KUKA KRL program: MyProgram_328().src

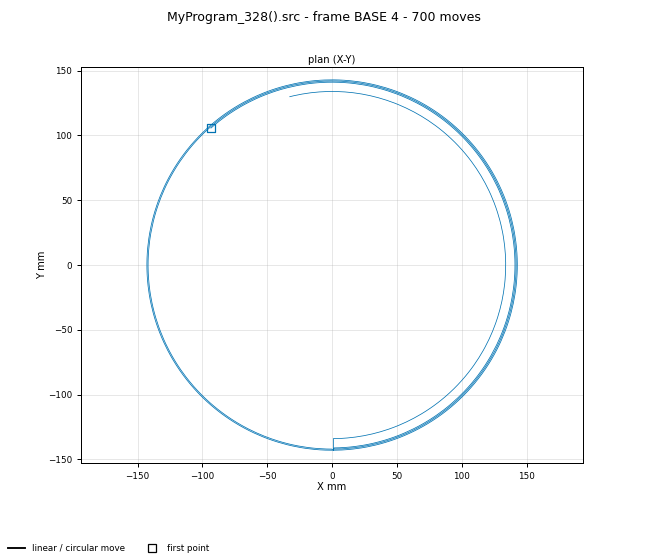
[picture p0: tool path of MyProgram_328().src in frame BASE 4, 700 of 700 moves have a stored position in this frame; points joined in program order, loops and branches not executed]
&ACCESS RVP
&REL 1
&PARAM TEMPLATE = C:\KRC\Roboter\Template\vorgabe
&PARAM EDITMASK = *
DEF MyProgram_328()
; ---- Setting reference (Base) ----
$BASE = BASE_DATA[4]

; --------------------------
; ---- Setting tool (TCP) ----
$TOOL = TOOL_DATA[3]
; --------------------------

$VEL.CP = VEL_APROX_PRINT
Startdeposition()
$VEL.CP = VEL_PRINT
LIN {X -93.4489,Y 105.68,Z 187,A 132.0784,B 2.4451,C 0.0422,E1 2.3432,E2 321.8422} C_DIS
LIN {X -90.1856,Y 108.4786,Z 187,A 130.186,B 2.4451,C 0.0397,E1 2.3473,E2 323.7515} C_DIS
LIN {X -86.5069,Y 111.4339,Z 187,A 128.2315,B 2.4451,C 0.0366,E1 2.3516,E2 325.7094} C_DIS
LIN {X -82.1262,Y 114.7007,Z 187,A 126.2266,B 2.4453,C 0.0324,E1 2.356,E2 327.6861} C_DIS
LIN {X -79.5267,Y 116.5186,Z 187,A 124.4196,B 2.4453,C 0.0324,E1 2.3603,E2 329.5564} C_DIS
LIN {X -74.9329,Y 119.5249,Z 187,A 121.6767,B 2.4453,C 0.0312,E1 2.3669,E2 332.3606} C_DIS
LIN {X -70.1382,Y 122.3996,Z 187,A 120.1865,B 2.4453,C 0.0253,E1 2.3703,E2 333.7537} C_DIS
LIN {X -67.2023,Y 124.0362,Z 187,A 118.5415,B 2.4453,C 0.0247,E1 2.3744,E2 335.4323} C_DIS
LIN {X -63.6582,Y 125.8895,Z 187,A 116.3136,B 2.4453,C 0.0253,E1 2.3802,E2 337.7328} C_DIS
LIN {X -58.7459,Y 128.2559,Z 187,A 114.739,B 2.4453,C 0.0203,E1 2.3839,E2 339.2278} C_DIS
LIN {X -55.245,Y 129.8038,Z 187,A 112.8056,B 2.4453,C 0.0204,E1 2.389,E2 341.2068} C_DIS
LIN {X -51.9085,Y 131.1741,Z 187,A 111.3758,B 2.4453,C 0.0189,E1 2.3927,E2 342.6315} C_DIS
LIN {X -45.9067,Y 133.3908,Z 187,A 108.9803,B 2.4454,C 0.016,E1 2.399,E2 345.0004} C_DIS
LIN {X -42.672,Y 134.4604,Z 187,A 107.5964,B 2.4454,C 0.015,E1 2.4027,E2 346.3836} C_DIS
LIN {X -39.1153,Y 135.5386,Z 187,A 105.5151,B 2.4454,C 0.0166,E1 2.4084,E2 348.5339} C_DIS
LIN {X -34.5458,Y 136.7738,Z 187,A 104.1224,B 2.4454,C 0.0131,E1 2.412,E2 349.8608} C_DIS
LIN {X -26.5142,Y 138.555,Z 187,A 100.5612,B 2.4454,C 0.0128,E1 2.4218,E2 353.4473} C_DIS
LIN {X -19.6263,Y 139.6976,Z 187,A 97.9243,B 2.4454,C 0.011,E1 2.4291,E2 356.0584} C_DIS
LIN {X -16.0676,Y 140.1526,Z 187,A 96.377,B 2.4454,C 0.0112,E1 2.4334,E2 357.6161} C_DIS
LIN {X -11.9745,Y 140.5601,Z 187,A 94.2351,B 2.4454,C 0.0135,E1 2.4395,E2 359.8147} C_DIS
LIN {X -7.2976,Y 140.8805,Z 187,A 92.8909,B 2.4454,C 0.0105,E1 2.4431,E2 361.0897} C_DIS
LIN {X -3.6531,Y 141.0223,Z 187,A 91.3608,B 2.4454,C 0.0109,E1 2.4474,E2 362.6252} C_DIS
LIN {X 0.7616,Y 141.0673,Z 187,A 89.5276,B 2.4454,C 0.0114,E1 2.4525,E2 364.4625} C_DIS
LIN {X 5.4307,Y 140.9647,Z 187,A 87.69,B 2.4454,C 0.0115,E1 2.4576,E2 366.2921} C_DIS
LIN {X 8.8719,Y 140.7901,Z 187,A 86.2614,B 2.4454,C 0.0122,E1 2.4616,E2 367.7237} C_DIS
LIN {X 13.2634,Y 140.4445,Z 187,A 84.4964,B 2.4454,C 0.0127,E1 2.4665,E2 369.4852} C_DIS
LIN {X 17.2396,Y 140.0128,Z 187,A 82.844,B 2.4454,C 0.0137,E1 2.4711,E2 371.1404} C_DIS
LIN {X 22.2924,Y 139.2984,Z 187,A 80.918,B 2.4454,C 0.014,E1 2.4764,E2 373.0478} C_DIS
LIN {X 24.9021,Y 138.8538,Z 187,A 79.8193,B 2.4454,C 0.0148,E1 2.4795,E2 374.1489} C_DIS
LIN {X 28.5165,Y 138.1573,Z 187,A 78.3416,B 2.4454,C 0.0158,E1 2.4835,E2 375.6241} C_DIS
LIN {X 32.2436,Y 137.3369,Z 187,A 76.8506,B 2.4454,C 0.0166,E1 2.4875,E2 377.1075} C_DIS
LIN {X 36.0345,Y 136.3894,Z 187,A 75.4608,B 2.4454,C 0.0167,E1 2.4913,E2 378.4724} C_DIS
LIN {X 38.942,Y 135.5894,Z 187,A 73.5871,B 2.4454,C 0.022,E1 2.4965,E2 380.4258} C_DIS
LIN {X 43.0848,Y 134.3286,Z 187,A 71.9887,B 2.4454,C 0.0227,E1 2.5007,E2 382.0041} C_DIS
LIN {X 46.6882,Y 133.1198,Z 187,A 70.8497,B 2.4454,C 0.0217,E1 2.5036,E2 383.093} C_DIS
LIN {X 49.6657,Y 132.037,Z 187,A 69.54,B 2.4454,C 0.0233,E1 2.507,E2 384.4053} C_DIS
LIN {X 53.4675,Y 130.5459,Z 187,A 67.9513,B 2.4454,C 0.0248,E1 2.5111,E2 385.9851} C_DIS
LIN {X 56.6566,Y 129.1935,Z 187,A 66.5966,B 2.4454,C 0.0262,E1 2.5146,E2 387.3331} C_DIS
LIN {X 59.5522,Y 127.883,Z 187,A 65.3245,B 2.4454,C 0.0278,E1 2.5178,E2 388.6026} C_DIS
LIN {X 62.4918,Y 126.472,Z 187,A 63.7782,B 2.4453,C 0.0311,E1 2.5218,E2 390.1762} C_DIS
LIN {X 65.3812,Y 125.0029,Z 187,A 62.7987,B 2.4453,C 0.0307,E1 2.5241,E2 391.1139} C_DIS
LIN {X 68.9963,Y 123.0467,Z 187,A 61.0451,B 2.4453,C 0.0337,E1 2.5284,E2 392.8779} C_DIS
LIN {X 72.7998,Y 120.8354,Z 187,A 59.2979,B 2.4452,C 0.0362,E1 2.5326,E2 394.6201} C_DIS
LIN {X 76.5853,Y 118.4724,Z 187,A 57.562,B 2.4452,C 0.0386,E1 2.5367,E2 396.3464} C_DIS
LIN {X 80.266,Y 116.0106,Z 187,A 55.7319,B 2.4452,C 0.0419,E1 2.5409,E2 398.1804} C_DIS
LIN {X 84.5184,Y 112.95,Z 187,A 53.7675,B 2.4451,C 0.0444,E1 2.5453,E2 400.1244} C_DIS
LIN {X 88.1752,Y 110.1193,Z 187,A 51.9494,B 2.4451,C 0.0474,E1 2.5493,E2 401.9351} C_DIS
LIN {X 91.0191,Y 107.7806,Z 187,A 50.5507,B 2.445,C 0.0495,E1 2.5523,E2 403.3218} C_DIS
LIN {X 94.151,Y 105.055,Z 187,A 48.609,B 2.4449,C 0.0547,E1 2.5564,E2 405.2955} C_DIS
LIN {X 97.1035,Y 102.3329,Z 187,A 47.579,B 2.4449,C 0.0535,E1 2.5584,E2 406.2504} C_DIS
LIN {X 100.7994,Y 98.6937,Z 187,A 45.3491,B 2.4448,C 0.0587,E1 2.5628,E2 408.496} C_DIS
LIN {X 103.7885,Y 95.5453,Z 187,A 43.6607,B 2.4447,C 0.0619,E1 2.566,E2 410.1752} C_DIS
LIN {X 106.7123,Y 92.2687,Z 187,A 41.9114,B 2.4446,C 0.0655,E1 2.5692,E2 411.9206} C_DIS
LIN {X 109.5484,Y 88.8835,Z 187,A 39.9522,B 2.4444,C 0.0708,E1 2.5727,E2 413.901} C_DIS
LIN {X 111.8638,Y 85.9509,Z 187,A 38.7393,B 2.4444,C 0.0719,E1 2.5747,E2 415.0758} C_DIS
LIN {X 114.5988,Y 82.2688,Z 187,A 37.005,B 2.4444,C 0.0752,E1 2.5776,E2 416.7942} C_DIS
LIN {X 117.0295,Y 78.7731,Z 187,A 35.3267,B 2.4442,C 0.0788,E1 2.5802,E2 418.4665} C_DIS
LIN {X 119.5196,Y 74.9413,Z 187,A 33.5491,B 2.4441,C 0.0827,E1 2.5829,E2 420.2346} C_DIS
LIN {X 121.8927,Y 71.0161,Z 187,A 31.7811,B 2.4439,C 0.0865,E1 2.5854,E2 421.9911} C_DIS
LIN {X 124.115,Y 67.0563,Z 187,A 30.0268,B 2.4438,C 0.0904,E1 2.5877,E2 423.7345} C_DIS
LIN {X 125.9818,Y 63.4769,Z 187,A 28.5834,B 2.4438,C 0.0929,E1 2.5895,E2 425.1532} C_DIS
LIN {X 127.4194,Y 60.5375,Z 187,A 27.2883,B 2.4436,C 0.096,E1 2.5911,E2 426.4444} C_DIS
LIN {X 128.9255,Y 57.2604,Z 187,A 25.9154,B 2.4435,C 0.099,E1 2.5927,E2 427.8061} C_DIS
LIN {X 130.3818,Y 53.8636,Z 187,A 24.5156,B 2.4433,C 0.1021,E1 2.5942,E2 429.1935} C_DIS
LIN {X 131.5987,Y 50.8162,Z 187,A 23.1723,B 2.4432,C 0.1057,E1 2.5956,E2 430.5386} C_DIS
LIN {X 132.8568,Y 47.4309,Z 187,A 21.8531,B 2.4431,C 0.1083,E1 2.5968,E2 431.8394} C_DIS
LIN {X 133.9409,Y 44.2758,Z 187,A 20.5533,B 2.4429,C 0.1115,E1 2.5979,E2 433.1327} C_DIS
LIN {X 135.1268,Y 40.5194,Z 187,A 18.45,B 2.4425,C 0.1201,E1 2.5997,E2 435.3016} C_DIS
LIN {X 136.5331,Y 35.4941,Z 187,A 17.0487,B 2.4425,C 0.1197,E1 2.6007,E2 436.6113} C_DIS
LIN {X 138.3504,Y 27.5676,Z 187,A 13.3763,B 2.4419,C 0.132,E1 2.6029,E2 440.3333} C_DIS
LIN {X 139.2135,Y 22.8091,Z 187,A 12.0869,B 2.4419,C 0.1316,E1 2.6034,E2 441.536} C_DIS
LIN {X 139.6764,Y 19.7745,Z 187,A 10.8655,B 2.4417,C 0.1349,E1 2.6039,E2 442.7547} C_DIS
LIN {X 140.0937,Y 16.5617,Z 187,A 9.6079,B 2.4416,C 0.138,E1 2.6043,E2 444.0055} C_DIS
LIN {X 140.5282,Y 12.3524,Z 187,A 7.8971,B 2.4413,C 0.1428,E1 2.6048,E2 445.7163} C_DIS
LIN {X 140.8206,Y 8.3778,Z 187,A 6.4549,B 2.4411,C 0.1458,E1 2.6051,E2 447.1363} C_DIS
LIN {X 141.0108,Y 4.0649,Z 187,A 4.8015,B 2.4409,C 0.1498,E1 2.6052,E2 448.7775} C_DIS
LIN {X 141.0688,Y 0.4654,Z 187,A 3.4438,B 2.4407,C 0.153,E1 2.6052,E2 450.1224} C_DIS
LIN {X 141.0307,Y -3.351,Z 187,A 2.023,B 2.4405,C 0.1563,E1 2.6052,E2 451.527} C_DIS
LIN {X 140.9079,Y -6.7536,Z 187,A 0.6135,B 2.4402,C 0.1604,E1 2.6051,E2 452.9409} C_DIS
LIN {X 140.6622,Y -10.7176,Z 187,A -0.8361,B 2.44,C 0.1635,E1 2.6048,E2 454.3699} C_DIS
LIN {X 140.3534,Y -14.2118,Z 187,A -2.3378,B 2.4397,C 0.1681,E1 2.6044,E2 455.8828} C_DIS
LIN {X 139.8712,Y -18.3453,Z 187,A -3.8669,B 2.4395,C 0.1715,E1 2.6039,E2 457.3917} C_DIS
LIN {X 139.3699,Y -21.831,Z 187,A -5.1458,B 2.4393,C 0.1741,E1 2.6033,E2 458.6513} C_DIS
LIN {X 138.8405,Y -24.9763,Z 187,A -6.4144,B 2.439,C 0.1775,E1 2.6027,E2 459.9172} C_DIS
LIN {X 137.7214,Y -30.5603,Z 187,A -8.657,B 2.4386,C 0.1832,E1 2.6015,E2 462.1522} C_DIS
LIN {X 136.491,Y -35.6537,Z 187,A -10.7762,B 2.4382,C 0.189,E1 2.6,E2 464.2718} C_DIS
LIN {X 135.288,Y -39.9714,Z 187,A -12.6689,B 2.4377,C 0.1946,E1 2.5985,E2 466.1754} C_DIS
LIN {X 134.115,Y -43.7528,Z 187,A -14.2718,B 2.4374,C 0.1989,E1 2.5972,E2 467.7789} C_DIS
LIN {X 132.7792,Y -47.6461,Z 187,A -15.5258,B 2.4374,C 0.1997,E1 2.596,E2 468.9781} C_DIS
LIN {X 131.393,Y -51.3455,Z 187,A -16.9763,B 2.4371,C 0.2026,E1 2.5946,E2 470.409} C_DIS
LIN {X 129.7181,Y -55.4433,Z 187,A -18.731,B 2.4367,C 0.207,E1 2.5927,E2 472.1593} C_DIS
LIN {X 126.8685,Y -61.688,Z 187,A -21.2796,B 2.4363,C 0.2121,E1 2.5898,E2 474.6779} C_DIS
LIN {X 122.4008,Y -70.1361,Z 187,A -24.8519,B 2.4356,C 0.2193,E1 2.5851,E2 478.2113} C_DIS
LIN {X 120.7802,Y -72.8911,Z 187,A -26.3212,B 2.4352,C 0.2239,E1 2.583,E2 479.705} C_DIS
LIN {X 118.2835,Y -76.8764,Z 187,A -28.2032,B 2.4348,C 0.2283,E1 2.5801,E2 481.5846} C_DIS
LIN {X 115.9942,Y -80.2896,Z 187,A -29.7454,B 2.4345,C 0.2312,E1 2.5777,E2 483.1109} C_DIS
LIN {X 112.5091,Y -85.1039,Z 187,A -31.8029,B 2.4343,C 0.2339,E1 2.5744,E2 485.1217} C_DIS
LIN {X 110.5589,Y -87.6229,Z 187,A -33.2922,B 2.4338,C 0.2385,E1 2.5718,E2 486.6387} C_DIS
LIN {X 107.5329,Y -91.3106,Z 187,A -35.3251,B 2.4333,C 0.2436,E1 2.5681,E2 488.6862} C_DIS
LIN {X 105.2436,Y -93.9402,Z 187,A -36.5934,B 2.4331,C 0.2455,E1 2.5658,E2 489.9354} C_DIS
LIN {X 101.7183,Y -97.7471,Z 187,A -39.1489,B 2.4323,C 0.2536,E1 2.5608,E2 492.5536} C_DIS
LIN {X 97.3968,Y -102.0531,Z 187,A -40.896,B 2.4323,C 0.2528,E1 2.5574,E2 494.203} C_DIS
LIN {X 92.0106,Y -106.9346,Z 187,A -43.3577,B 2.4322,C 0.2547,E1 2.5525,E2 496.5995} C_DIS
LIN {X 88.677,Y -109.7149,Z 187,A -45.5587,B 2.4314,C 0.2615,E1 2.5476,E2 498.8623} C_DIS
LIN {X 86.1521,Y -111.7089,Z 187,A -47.2607,B 2.4309,C 0.267,E1 2.5437,E2 500.6194} C_DIS
LIN {X 81.5208,Y -115.132,Z 187,A -48.6174,B 2.4312,C 0.2635,E1 2.5409,E2 501.8429} C_DIS
LIN {X 79.0495,Y -116.8424,Z 187,A -50.4786,B 2.4305,C 0.2706,E1 2.5364,E2 503.7933} C_DIS
LIN {X 75.3103,Y -119.2862,Z 187,A -51.9221,B 2.4305,C 0.2707,E1 2.5331,E2 505.1872} C_DIS
LIN {X 71.0161,Y -121.8927,Z 187,A -53.8333,B 2.4302,C 0.2729,E1 2.5285,E2 507.0822} C_DIS
LIN {X 67.0764,Y -124.1042,Z 187,A -55.6212,B 2.4299,C 0.2753,E1 2.5242,E2 508.8648} C_DIS
LIN {X 63.1985,Y -126.1233,Z 187,A -57.2403,B 2.4298,C 0.2767,E1 2.5202,E2 510.4636} C_DIS
LIN {X 56.1606,Y -129.408,Z 187,A -60.0745,B 2.4296,C 0.2786,E1 2.5131,E2 513.2555} C_DIS
LIN {X 51.9792,Y -131.1459,Z 187,A -62.1004,B 2.4291,C 0.2822,E1 2.5078,E2 515.3088} C_DIS
LIN {X 48.5186,Y -132.4646,Z 187,A -63.7676,B 2.4288,C 0.2851,E1 2.5034,E2 516.9996} C_DIS
LIN {X 44.3169,Y -133.9273,Z 187,A -65.3456,B 2.4288,C 0.2854,E1 2.4993,E2 518.5469} C_DIS
LIN {X 40.4578,Y -135.1456,Z 187,A -67.0119,B 2.4285,C 0.2873,E1 2.4948,E2 520.2175} C_DIS
LIN {X 36.0324,Y -136.39,Z 187,A -68.8114,B 2.4284,C 0.2885,E1 2.49,E2 522.0087} C_DIS
LIN {X 31.8028,Y -137.438,Z 187,A -70.552,B 2.4282,C 0.2898,E1 2.4852,E2 523.7464} C_DIS
LIN {X 27.8459,Y -138.2937,Z 187,A -72.1648,B 2.4282,C 0.2909,E1 2.4808,E2 525.3558} C_DIS
LIN {X 24.2043,Y -138.9786,Z 187,A -74.473,B 2.4274,C 0.2972,E1 2.4742,E2 527.7761} C_DIS
LIN {X 17.7076,Y -139.9548,Z 187,A -76.3709,B 2.4278,C 0.2937,E1 2.4692,E2 529.5691} C_DIS
LIN {X 13.6314,Y -140.4091,Z 187,A -77.9481,B 2.4278,C 0.2939,E1 2.4648,E2 531.1348} C_DIS
LIN {X 9.8054,Y -140.7288,Z 187,A -79.5631,B 2.4276,C 0.2949,E1 2.4603,E2 532.7584} C_DIS
LIN {X 5.6236,Y -140.9572,Z 187,A -81.1799,B 2.4276,C 0.2949,E1 2.4558,E2 534.3642} C_DIS
LIN {X 1.6647,Y -141.0612,Z 187,A -82.8613,B 2.4276,C 0.2958,E1 2.4511,E2 536.0567} C_DIS
LIN {X 1.6647,Y -141.0612,Z 187,A -82.8613,B 2.4276,C 0.2958,E1 2.4511,E2 536.0567} C_DIS
Enddeposition()
LIN {X 0.9996,Y -141.963,Z 187,A -82.7924,B 2.4278,C 0.2951,E1 2.4515,E2 535.9704} C_DIS
Startdeposition()
$VEL.CP = VEL_PRINT
LIN {X 3.7682,Y -141.9191,Z 187,A -81.2714,B 2.4281,C 0.2923,E1 2.4559,E2 534.3919} C_DIS
LIN {X 7.2589,Y -141.7833,Z 187,A -79.8823,B 2.4281,C 0.292,E1 2.4598,E2 533.005} C_DIS
LIN {X 11.0857,Y -141.5374,Z 187,A -78.324,B 2.4282,C 0.2913,E1 2.4641,E2 531.4445} C_DIS
LIN {X 14.9868,Y -141.1758,Z 187,A -76.8976,B 2.4282,C 0.2915,E1 2.468,E2 530.039} C_DIS
LIN {X 17.882,Y -140.8393,Z 187,A -75.3634,B 2.4285,C 0.2885,E1 2.4724,E2 528.4534} C_DIS
LIN {X 23.036,Y -140.0878,Z 187,A -73.5358,B 2.4285,C 0.2891,E1 2.4774,E2 526.6635} C_DIS
LIN {X 26.407,Y -139.4914,Z 187,A -72.2818,B 2.4285,C 0.289,E1 2.4808,E2 525.4268} C_DIS
LIN {X 29.7911,Y -138.8079,Z 187,A -70.7974,B 2.4287,C 0.2873,E1 2.4849,E2 523.9287} C_DIS
LIN {X 32.6858,Y -138.1561,Z 187,A -69.705,B 2.4287,C 0.287,E1 2.4878,E2 522.8505} C_DIS
LIN {X 36.0579,Y -137.3143,Z 187,A -68.3438,B 2.4288,C 0.2861,E1 2.4915,E2 521.4943} C_DIS
LIN {X 39.1204,Y -136.4746,Z 187,A -66.8529,B 2.4291,C 0.2834,E1 2.4956,E2 519.973} C_DIS
LIN {X 43.2015,Y -135.2357,Z 187,A -65.3089,B 2.4291,C 0.2829,E1 2.4997,E2 518.4528} C_DIS
LIN {X 47.5675,Y -133.7639,Z 187,A -63.4225,B 2.4295,C 0.2807,E1 2.5047,E2 516.5614} C_DIS
LIN {X 51.1458,Y -132.4359,Z 187,A -62.0665,B 2.4295,C 0.2803,E1 2.5082,E2 515.2304} C_DIS
LIN {X 53.7562,Y -131.3996,Z 187,A -60.7366,B 2.4298,C 0.2774,E1 2.5117,E2 513.8721} C_DIS
LIN {X 56.7664,Y -130.1262,Z 187,A -59.2192,B 2.4302,C 0.2743,E1 2.5156,E2 512.3256} C_DIS
LIN {X 60.3683,Y -128.4969,Z 187,A -57.8944,B 2.4302,C 0.2741,E1 2.5189,E2 511.0381} C_DIS
LIN {X 63.9328,Y -126.7593,Z 187,A -56.289,B 2.4305,C 0.2718,E1 2.5229,E2 509.4308} C_DIS
LIN {X 68.2838,Y -124.4711,Z 187,A -54.4459,B 2.4307,C 0.27,E1 2.5274,E2 507.6063} C_DIS
LIN {X 71.2977,Y -122.7693,Z 187,A -52.7218,B 2.4312,C 0.2653,E1 2.5317,E2 505.8348} C_DIS
LIN {X 75.1294,Y -120.4624,Z 187,A -50.6328,B 2.4317,C 0.2601,E1 2.5367,E2 503.7041} C_DIS
LIN {X 80.5629,Y -116.8987,Z 187,A -49.0053,B 2.4314,C 0.2635,E1 2.5402,E2 502.2154} C_DIS
LIN {X 84.7135,Y -113.9265,Z 187,A -46.767,B 2.4319,C 0.2584,E1 2.5453,E2 499.9506} C_DIS
LIN {X 88.639,Y -110.9,Z 187,A -44.9104,B 2.4322,C 0.2559,E1 2.5494,E2 498.1126} C_DIS
LIN {X 92.22,Y -107.9408,Z 187,A -43.2469,B 2.4324,C 0.254,E1 2.5529,E2 496.4773} C_DIS
LIN {X 95.9781,Y -104.6128,Z 187,A -40.9372,B 2.433,C 0.2476,E1 2.5577,E2 494.1263} C_DIS
LIN {X 98.5673,Y -102.1771,Z 187,A -39.7798,B 2.4331,C 0.247,E1 2.56,E2 493.0066} C_DIS
LIN {X 101.6156,Y -99.1464,Z 187,A -38.1008,B 2.4334,C 0.2438,E1 2.5633,E2 491.3341} C_DIS
LIN {X 104.7827,Y -95.7932,Z 187,A -36.4189,B 2.4337,C 0.2413,E1 2.5664,E2 489.6758} C_DIS
LIN {X 107.0817,Y -93.2155,Z 187,A -34.6604,B 2.4343,C 0.2352,E1 2.5698,E2 487.8652} C_DIS
LIN {X 109.8305,Y -89.9605,Z 187,A -33.3443,B 2.4343,C 0.2347,E1 2.572,E2 486.6041} C_DIS
LIN {X 112.7503,Y -86.2727,Z 187,A -31.4726,B 2.4347,C 0.2306,E1 2.5752,E2 484.7347} C_DIS
LIN {X 115.5827,Y -82.4395,Z 187,A -29.7495,B 2.435,C 0.2278,E1 2.578,E2 483.0379} C_DIS
LIN {X 118.0467,Y -78.8707,Z 187,A -28.0529,B 2.4353,C 0.2241,E1 2.5807,E2 481.3474} C_DIS
LIN {X 120.4789,Y -75.103,Z 187,A -26.318,B 2.4357,C 0.2203,E1 2.5832,E2 479.6215} C_DIS
LIN {X 122.8161,Y -71.2168,Z 187,A -24.7349,B 2.4359,C 0.2179,E1 2.5854,E2 478.0712} C_DIS
LIN {X 125.4596,Y -66.4467,Z 187,A -22.5256,B 2.4364,C 0.2123,E1 2.5884,E2 475.859} C_DIS
LIN {X 127.0868,Y -63.2792,Z 187,A -21.155,B 2.4366,C 0.2092,E1 2.5901,E2 474.4964} C_DIS
LIN {X 128.6491,Y -60.039,Z 187,A -19.6284,B 2.437,C 0.2048,E1 2.592,E2 472.9584} C_DIS
LIN {X 130.7091,Y -55.4144,Z 187,A -17.9178,B 2.4372,C 0.2024,E1 2.5938,E2 471.2921} C_DIS
LIN {X 132.1546,Y -51.8693,Z 187,A -16.3795,B 2.4376,C 0.1984,E1 2.5954,E2 469.7535} C_DIS
LIN {X 134.6378,Y -45.0306,Z 187,A -13.8601,B 2.4379,C 0.1943,E1 2.5977,E2 467.2891} C_DIS
LIN {X 135.6936,Y -41.7415,Z 187,A -12.2862,B 2.4383,C 0.1889,E1 2.5991,E2 465.6896} C_DIS
LIN {X 136.6561,Y -38.4741,Z 187,A -10.6448,B 2.4388,C 0.1828,E1 2.6004,E2 464.0107} C_DIS
LIN {X 137.6676,Y -34.6814,Z 187,A -9.4864,B 2.4388,C 0.1822,E1 2.6011,E2 462.9095} C_DIS
LIN {X 138.626,Y -30.6336,Z 187,A -7.7706,B 2.4392,C 0.1773,E1 2.6022,E2 461.1875} C_DIS
LIN {X 139.3977,Y -26.8975,Z 187,A -6.4337,B 2.4394,C 0.1748,E1 2.6029,E2 459.877} C_DIS
LIN {X 140.0385,Y -23.3314,Z 187,A -5.0733,B 2.4396,C 0.1717,E1 2.6035,E2 458.5294} C_DIS
LIN {X 140.6556,Y -19.2805,Z 187,A -3.4323,B 2.4399,C 0.1672,E1 2.6042,E2 456.8891} C_DIS
LIN {X 141.1483,Y -15.2421,Z 187,A -1.975,B 2.4401,C 0.1642,E1 2.6046,E2 455.4556} C_DIS
LIN {X 141.4775,Y -11.8026,Z 187,A -0.6039,B 2.4403,C 0.1605,E1 2.605,E2 454.0868} C_DIS
LIN {X 141.7785,Y -7.3542,Z 187,A 1.0076,B 2.4406,C 0.1571,E1 2.6053,E2 452.4994} C_DIS
LIN {X 141.9161,Y -3.8773,Z 187,A 2.4541,B 2.4408,C 0.1528,E1 2.6053,E2 451.0464} C_DIS
LIN {X 141.9682,Y 0.508,Z 187,A 4.1072,B 2.4411,C 0.1489,E1 2.6054,E2 449.4078} C_DIS
LIN {X 141.9065,Y 4.2199,Z 187,A 5.523,B 2.4413,C 0.1454,E1 2.6054,E2 448.0023} C_DIS
LIN {X 141.7092,Y 8.5854,Z 187,A 7.0861,B 2.4415,C 0.1422,E1 2.6051,E2 446.465} C_DIS
LIN {X 141.4746,Y 11.8375,Z 187,A 8.4459,B 2.4417,C 0.1381,E1 2.6048,E2 445.0986} C_DIS
LIN {X 141.0538,Y 16.1086,Z 187,A 10.1489,B 2.442,C 0.1336,E1 2.6043,E2 443.3986} C_DIS
LIN {X 140.5408,Y 20.0852,Z 187,A 11.5878,B 2.4421,C 0.1306,E1 2.6038,E2 441.9826} C_DIS
LIN {X 139.991,Y 23.6157,Z 187,A 13.0025,B 2.4423,C 0.1269,E1 2.6031,E2 440.5708} C_DIS
LIN {X 139.0168,Y 28.8045,Z 187,A 15.0092,B 2.4426,C 0.1221,E1 2.602,E2 438.5795} C_DIS
LIN {X 138.0808,Y 32.9981,Z 187,A 16.6182,B 2.4427,C 0.1184,E1 2.601,E2 436.9862} C_DIS
LIN {X 137.2031,Y 36.4748,Z 187,A 17.9412,B 2.4429,C 0.1155,E1 2.6001,E2 435.679} C_DIS
LIN {X 136.3607,Y 39.5094,Z 187,A 19.3511,B 2.4431,C 0.1109,E1 2.599,E2 434.25} C_DIS
LIN {X 134.8365,Y 44.4339,Z 187,A 21.0397,B 2.4431,C 0.1087,E1 2.5976,E2 432.6123} C_DIS
LIN {X 133.687,Y 47.7808,Z 187,A 22.431,B 2.4433,C 0.1052,E1 2.5964,E2 431.2252} C_DIS
LIN {X 132.5412,Y 50.8749,Z 187,A 23.6494,B 2.4435,C 0.1026,E1 2.5952,E2 430.0213} C_DIS
LIN {X 131.0962,Y 54.4875,Z 187,A 25.1666,B 2.4436,C 0.0989,E1 2.5936,E2 428.5103} C_DIS
LIN {X 129.7867,Y 57.5383,Z 187,A 26.5247,B 2.4438,C 0.0953,E1 2.5921,E2 427.1493} C_DIS
LIN {X 128.2461,Y 60.8941,Z 187,A 27.9417,B 2.4438,C 0.0921,E1 2.5904,E2 425.7414} C_DIS
LIN {X 126.7611,Y 63.9292,Z 187,A 29.2664,B 2.444,C 0.0889,E1 2.5888,E2 424.4213} C_DIS
LIN {X 124.8445,Y 67.5992,Z 187,A 30.9033,B 2.4441,C 0.085,E1 2.5866,E2 422.7884} C_DIS
LIN {X 122.644,Y 71.514,Z 187,A 32.6528,B 2.4443,C 0.0811,E1 2.5842,E2 421.0466} C_DIS
LIN {X 120.3764,Y 75.2676,Z 187,A 34.287,B 2.4443,C 0.0779,E1 2.5818,E2 419.4295} C_DIS
LIN {X 117.9973,Y 78.9446,Z 187,A 35.9633,B 2.4445,C 0.0744,E1 2.5793,E2 417.7645} C_DIS
LIN {X 115.4017,Y 82.6927,Z 187,A 37.7059,B 2.4445,C 0.0709,E1 2.5765,E2 416.0342} C_DIS
LIN {X 112.7821,Y 86.2311,Z 187,A 39.4389,B 2.4447,C 0.0672,E1 2.5736,E2 414.3063} C_DIS
LIN {X 110.0375,Y 89.7071,Z 187,A 41.1027,B 2.4447,C 0.0641,E1 2.5707,E2 412.6582} C_DIS
LIN {X 107.4472,Y 92.794,Z 187,A 42.6833,B 2.4449,C 0.0609,E1 2.5678,E2 411.0833} C_DIS
LIN {X 104.407,Y 96.2019,Z 187,A 44.4152,B 2.4449,C 0.0578,E1 2.5646,E2 409.3654} C_DIS
LIN {X 101.4157,Y 99.3502,Z 187,A 46.1356,B 2.445,C 0.0544,E1 2.5613,E2 407.6489} C_DIS
LIN {X 98.1632,Y 102.5651,Z 187,A 47.6842,B 2.445,C 0.0529,E1 2.5583,E2 406.1382} C_DIS
LIN {X 95.5959,Y 104.9624,Z 187,A 49.2623,B 2.4451,C 0.0489,E1 2.555,E2 404.5394} C_DIS
LIN {X 92.3606,Y 107.8205,Z 187,A 50.9361,B 2.4451,C 0.046,E1 2.5515,E2 402.8743} C_DIS
LIN {X 89.3733,Y 110.3091,Z 187,A 52.4532,B 2.4452,C 0.0435,E1 2.5482,E2 401.3637} C_DIS
LIN {X 85.9012,Y 113.0344,Z 187,A 54.1813,B 2.4452,C 0.0406,E1 2.5444,E2 399.6424} C_DIS
LIN {X 82.3582,Y 115.6409,Z 187,A 55.8678,B 2.4453,C 0.0382,E1 2.5406,E2 397.9673} C_DIS
LIN {X 78.849,Y 118.0612,Z 187,A 57.5179,B 2.4453,C 0.0358,E1 2.5368,E2 396.3261} C_DIS
LIN {X 75.3466,Y 120.3273,Z 187,A 59.1625,B 2.4453,C 0.0334,E1 2.5329,E2 394.6866} C_DIS
LIN {X 71.5652,Y 122.614,Z 187,A 60.9314,B 2.4454,C 0.0307,E1 2.5287,E2 392.9196} C_DIS
LIN {X 67.5831,Y 124.8533,Z 187,A 62.5878,B 2.4454,C 0.0293,E1 2.5247,E2 391.2871} C_DIS
LIN {X 65.0121,Y 126.2098,Z 187,A 63.8486,B 2.4454,C 0.027,E1 2.5215,E2 390.0153} C_DIS
LIN {X 61.8211,Y 127.8032,Z 187,A 65.2354,B 2.4454,C 0.0254,E1 2.5181,E2 388.6354} C_DIS
LIN {X 58.2382,Y 129.4737,Z 187,A 66.5719,B 2.4454,C 0.0251,E1 2.5147,E2 387.3317} C_DIS
LIN {X 55.7537,Y 130.5641,Z 187,A 67.8714,B 2.4455,C 0.0224,E1 2.5113,E2 386.0066} C_DIS
LIN {X 51.9672,Y 132.1165,Z 187,A 69.3282,B 2.4455,C 0.0217,E1 2.5076,E2 384.5747} C_DIS
LIN {X 48.52,Y 133.4205,Z 187,A 70.6667,B 2.4455,C 0.021,E1 2.5042,E2 383.2552} C_DIS
LIN {X 42.9455,Y 135.3175,Z 187,A 73.8187,B 2.4455,C 0.0135,E1 2.4955,E2 380.0055} C_DIS
LIN {X 37.6109,Y 136.8975,Z 187,A 75.6157,B 2.4455,C 0.0144,E1 2.4908,E2 378.2661} C_DIS
LIN {X 32.6143,Y 138.1733,Z 187,A 77.409,B 2.4455,C 0.0144,E1 2.4861,E2 376.5098} C_DIS
LIN {X 29.0269,Y 138.9716,Z 187,A 78.9989,B 2.4455,C 0.0127,E1 2.4817,E2 374.9068} C_DIS
LIN {X 25.5257,Y 139.6561,Z 187,A 80.1674,B 2.4455,C 0.0134,E1 2.4786,E2 373.7728} C_DIS
LIN {X 22.4562,Y 140.1835,Z 187,A 81.7525,B 2.4455,C 0.0106,E1 2.4741,E2 372.1469} C_DIS
LIN {X 17.6812,Y 140.8656,Z 187,A 83.5823,B 2.4455,C 0.0103,E1 2.469,E2 370.3325} C_DIS
LIN {X 13.7164,Y 141.3048,Z 187,A 85.0418,B 2.4455,C 0.0105,E1 2.465,E2 368.8924} C_DIS
LIN {X 10.2703,Y 141.597,Z 187,A 86.3842,B 2.4455,C 0.0102,E1 2.4613,E2 367.5571} C_DIS
LIN {X 7.1493,Y 141.7888,Z 187,A 87.7138,B 2.4455,C 0.0094,E1 2.4576,E2 366.2196} C_DIS
LIN {X 2.9737,Y 141.9392,Z 187,A 89.4396,B 2.4455,C 0.0088,E1 2.4527,E2 364.4895} C_DIS
LIN {X -0.7732,Y 141.9669,Z 187,A 90.954,B 2.4455,C 0.0085,E1 2.4485,E2 362.9754} C_DIS
LIN {X -5.5262,Y 141.8614,Z 187,A 92.7703,B 2.4455,C 0.009,E1 2.4434,E2 361.1728} C_DIS
LIN {X -9.8597,Y 141.6269,Z 187,A 94.4629,B 2.4455,C 0.0093,E1 2.4387,E2 359.4883} C_DIS
LIN {X -13.6559,Y 141.3106,Z 187,A 96.1386,B 2.4455,C 0.0087,E1 2.434,E2 357.796} C_DIS
LIN {X -18.1954,Y 140.7982,Z 187,A 97.9544,B 2.4455,C 0.0091,E1 2.429,E2 355.9846} C_DIS
LIN {X -22.019,Y 140.2512,Z 187,A 99.9681,B 2.4455,C 0.0072,E1 2.4233,E2 353.9145} C_DIS
LIN {X -26.3023,Y 139.5114,Z 187,A 101.2219,B 2.4455,C 0.0104,E1 2.42,E2 352.7246} C_DIS
LIN {X -29.1917,Y 138.9373,Z 187,A 102.516,B 2.4455,C 0.0104,E1 2.4164,E2 351.418} C_DIS
LIN {X -32.657,Y 138.163,Z 187,A 104.0144,B 2.4455,C 0.0107,E1 2.4123,E2 349.9122} C_DIS
LIN {X -36.3809,Y 137.2281,Z 187,A 105.8057,B 2.4455,C 0.0104,E1 2.4074,E2 348.0913} C_DIS
LIN {X -39.7779,Y 136.2821,Z 187,A 106.9762,B 2.4455,C 0.0125,E1 2.4043,E2 346.9533} C_DIS
LIN {X -43.7202,Y 135.07,Z 187,A 108.7525,B 2.4455,C 0.0131,E1 2.3995,E2 345.164} C_DIS
LIN {X -50.6272,Y 132.6373,Z 187,A 111.7286,B 2.4455,C 0.0154,E1 2.3917,E2 342.1872} C_DIS
LIN {X -54.3321,Y 131.1611,Z 187,A 113.1961,B 2.4455,C 0.0175,E1 2.388,E2 340.7384} C_DIS
LIN {X -57.7103,Y 129.7098,Z 187,A 114.7724,B 2.4455,C 0.0186,E1 2.3839,E2 339.1514} C_DIS
LIN {X -60.7714,Y 128.3047,Z 187,A 116.4131,B 2.4455,C 0.0188,E1 2.3797,E2 337.4761} C_DIS
LIN {X -63.6843,Y 126.8858,Z 187,A 117.5622,B 2.4455,C 0.021,E1 2.3768,E2 336.348} C_DIS
LIN {X -67.4063,Y 124.9482,Z 187,A 119.3288,B 2.4455,C 0.0227,E1 2.3724,E2 334.5732} C_DIS
LIN {X -70.536,Y 123.2085,Z 187,A 120.9137,B 2.4455,C 0.0239,E1 2.3685,E2 332.9716} C_DIS
LIN {X -74.8507,Y 120.6359,Z 187,A 122.9065,B 2.4455,C 0.0268,E1 2.3638,E2 330.9845} C_DIS
LIN {X -78.7501,Y 118.1272,Z 187,A 124.8088,B 2.4455,C 0.0293,E1 2.3593,E2 329.0797} C_DIS
LIN {X -82.3891,Y 115.6187,Z 187,A 126.694,B 2.4455,C 0.0316,E1 2.355,E2 327.1828} C_DIS
LIN {X -86.1482,Y 112.8455,Z 187,A 128.5791,B 2.4454,C 0.0346,E1 2.3508,E2 325.299} C_DIS
LIN {X -89.5032,Y 110.2042,Z 187,A 130.4211,B 2.4454,C 0.0371,E1 2.3467,E2 323.4433} C_DIS
LIN {X -93.0071,Y 107.2636,Z 187,A 132.1594,B 2.4453,C 0.0406,E1 2.3431,E2 321.7199} C_DIS
LIN {X -95.6368,Y 104.9252,Z 187,A 133.7545,B 2.4453,C 0.0426,E1 2.3397,E2 320.1036} C_DIS
LIN {X -98.7853,Y 101.966,Z 187,A 135.5669,B 2.4452,C 0.0456,E1 2.336,E2 318.2837} C_DIS
LIN {X -101.5357,Y 99.2279,Z 187,A 137.2404,B 2.4452,C 0.0482,E1 2.3327,E2 316.5978} C_DIS
LIN {X -104.3309,Y 96.2847,Z 187,A 139.0136,B 2.4451,C 0.051,E1 2.3293,E2 314.8086} C_DIS
LIN {X -107.6788,Y 92.5251,Z 187,A 141.0456,B 2.445,C 0.0552,E1 2.3256,E2 312.778} C_DIS
LIN {X -110.2091,Y 89.4973,Z 187,A 142.77,B 2.445,C 0.0581,E1 2.3225,E2 311.0379} C_DIS
LIN {X -113.0558,Y 85.8731,Z 187,A 144.4305,B 2.4448,C 0.0627,E1 2.3197,E2 309.4042} C_DIS
LIN {X -115.947,Y 81.9263,Z 187,A 146.6612,B 2.4448,C 0.0664,E1 2.316,E2 307.1423} C_DIS
LIN {X -117.5624,Y 79.5907,Z 187,A 147.9369,B 2.4446,C 0.0686,E1 2.3139,E2 305.8508} C_DIS
LIN {X -119.9532,Y 75.94,Z 187,A 149.8296,B 2.4446,C 0.0723,E1 2.311,E2 303.9425} C_DIS
LIN {X -122.4267,Y 71.8841,Z 187,A 151.805,B 2.4444,C 0.0767,E1 2.3082,E2 301.961} C_DIS
LIN {X -124.6117,Y 68.026,Z 187,A 153.5249,B 2.4443,C 0.0812,E1 2.3059,E2 300.2514} C_DIS
LIN {X -126.197,Y 65.0371,Z 187,A 155.1662,B 2.4442,C 0.0838,E1 2.3037,E2 298.5755} C_DIS
LIN {X -127.8502,Y 61.7227,Z 187,A 156.6552,B 2.444,C 0.0875,E1 2.3019,E2 297.0882} C_DIS
LIN {X -129.4019,Y 58.3988,Z 187,A 158.1848,B 2.444,C 0.0912,E1 2.3001,E2 295.5534} C_DIS
LIN {X -130.9979,Y 54.723,Z 187,A 159.7031,B 2.4437,C 0.0956,E1 2.2984,E2 294.0491} C_DIS
LIN {X -132.2138,Y 51.7171,Z 187,A 161.3539,B 2.4437,C 0.0981,E1 2.2967,E2 292.3548} C_DIS
LIN {X -133.6411,Y 47.9081,Z 187,A 162.9786,B 2.4435,C 0.1024,E1 2.2951,E2 290.7336} C_DIS
LIN {X -134.6713,Y 44.9302,Z 187,A 164.4028,B 2.4433,C 0.1054,E1 2.2938,E2 289.2904} C_DIS
LIN {X -135.768,Y 41.4984,Z 187,A 165.9228,B 2.4432,C 0.1091,E1 2.2926,E2 287.7628} C_DIS
LIN {X -136.7761,Y 38.0449,Z 187,A 167.4839,B 2.443,C 0.1127,E1 2.2914,E2 286.1885} C_DIS
LIN {X -137.9061,Y 33.7228,Z 187,A 169.4221,B 2.4428,C 0.1173,E1 2.29,E2 284.2339} C_DIS
LIN {X -139.805,Y 24.6939,Z 187,A 172.8607,B 2.4422,C 0.1283,E1 2.2881,E2 280.8355} C_DIS
LIN {X -140.4475,Y 20.7386,Z 187,A 175.1058,B 2.4421,C 0.1312,E1 2.2871,E2 278.5092} C_DIS
LIN {X -140.8929,Y 17.4571,Z 187,A 176.5678,B 2.4419,C 0.1346,E1 2.2865,E2 277.0315} C_DIS
LIN {X -141.3104,Y 13.6576,Z 187,A 177.9513,B 2.4416,C 0.1393,E1 2.2862,E2 275.6699} C_DIS
LIN {X -141.5316,Y 11.1627,Z 187,A 179.2339,B 2.4416,C 0.1414,E1 2.2859,E2 274.3522} C_DIS
LIN {X -141.7436,Y 8.0273,Z 187,A -179.3993,B 2.4413,C 0.1448,E1 2.2856,E2 272.9731} C_DIS
LIN {X -141.9294,Y 3.3985,Z 187,A -177.394,B 2.441,C 0.1497,E1 2.2854,E2 270.9508} C_DIS
LIN {X -141.9653,Y -1.0663,Z 187,A -175.5455,B 2.4407,C 0.1546,E1 2.2854,E2 269.0972} C_DIS
LIN {X -141.8675,Y -5.3683,Z 187,A -173.8566,B 2.4404,C 0.1596,E1 2.2856,E2 267.4158} C_DIS
LIN {X -141.6419,Y -9.655,Z 187,A -171.8203,B 2.4401,C 0.1637,E1 2.2859,E2 265.34} C_DIS
LIN {X -141.1197,Y -15.5075,Z 187,A -169.3476,B 2.4397,C 0.17,E1 2.2866,E2 262.8551} C_DIS
LIN {X -140.5823,Y -19.795,Z 187,A -167.6331,B 2.4393,C 0.175,E1 2.2872,E2 261.1456} C_DIS
LIN {X -140.0836,Y -23.0608,Z 187,A -166.1046,B 2.4391,C 0.1781,E1 2.2879,E2 259.5915} C_DIS
LIN {X -138.9037,Y -29.3472,Z 187,A -163.3411,B 2.4386,C 0.1848,E1 2.2894,E2 256.8049} C_DIS
LIN {X -138.0745,Y -33.0242,Z 187,A -161.768,B 2.4383,C 0.1887,E1 2.2904,E2 255.2255} C_DIS
LIN {X -137.1868,Y -36.536,Z 187,A -160.1642,B 2.438,C 0.1923,E1 2.2915,E2 253.6032} C_DIS
LIN {X -136.0472,Y -40.5803,Z 187,A -158.3514,B 2.4377,C 0.1965,E1 2.2929,E2 251.7754} C_DIS
LIN {X -134.8365,Y -44.4339,Z 187,A -156.6444,B 2.4374,C 0.2006,E1 2.2944,E2 250.0587} C_DIS
LIN {X -133.862,Y -47.2942,Z 187,A -155.2575,B 2.4371,C 0.2034,E1 2.2957,E2 248.6496} C_DIS
LIN {X -132.4832,Y -51.0242,Z 187,A -153.8732,B 2.4367,C 0.2081,E1 2.297,E2 247.296} C_DIS
LIN {X -131.1245,Y -54.4197,Z 187,A -152.1482,B 2.4365,C 0.2112,E1 2.2989,E2 245.5377} C_DIS
LIN {X -129.7648,Y -57.5874,Z 187,A -150.8505,B 2.4361,C 0.215,E1 2.3003,E2 244.2533} C_DIS
LIN {X -128.3173,Y -60.745,Z 187,A -149.1765,B 2.4359,C 0.2177,E1 2.3023,E2 242.5427} C_DIS
LIN {X -126.6965,Y -64.056,Z 187,A -147.6242,B 2.4356,C 0.2212,E1 2.3043,E2 240.9821} C_DIS
LIN {X -125.4667,Y -66.4333,Z 187,A -146.3905,B 2.4354,C 0.2233,E1 2.3059,E2 239.7277} C_DIS
LIN {X -123.2211,Y -70.5139,Z 187,A -144.4516,B 2.435,C 0.2276,E1 2.3086,E2 237.7813} C_DIS
LIN {X -121.0422,Y -74.1916,Z 187,A -142.6392,B 2.4346,C 0.2314,E1 2.3112,E2 235.9574} C_DIS
LIN {X -119.0867,Y -77.2915,Z 187,A -141.0822,B 2.4343,C 0.2345,E1 2.3136,E2 234.3901} C_DIS
LIN {X -116.603,Y -80.9898,Z 187,A -139.1606,B 2.434,C 0.2381,E1 2.3166,E2 232.4519} C_DIS
LIN {X -112.7149,Y -86.319,Z 187,A -136.4228,B 2.4334,C 0.2437,E1 2.3212,E2 229.7043} C_DIS
LIN {X -110.1029,Y -89.6272,Z 187,A -134.5808,B 2.4331,C 0.2467,E1 2.3245,E2 227.8431} C_DIS
LIN {X -106.6874,Y -93.6675,Z 187,A -132.334,B 2.4327,C 0.2507,E1 2.3286,E2 225.5812} C_DIS
LIN {X -103.8762,Y -96.7746,Z 187,A -130.6176,B 2.4324,C 0.2539,E1 2.3318,E2 223.8615} C_DIS
LIN {X -100.6604,Y -100.1154,Z 187,A -128.9128,B 2.432,C 0.2581,E1 2.3351,E2 222.1802} C_DIS
LIN {X -97.5447,Y -103.1536,Z 187,A -126.8353,B 2.4317,C 0.2601,E1 2.3394,E2 220.0581} C_DIS
LIN {X -94.2288,Y -106.1914,Z 187,A -125.112,B 2.4314,C 0.2636,E1 2.3429,E2 218.3478} C_DIS
LIN {X -91.3588,Y -108.6701,Z 187,A -123.3568,B 2.4312,C 0.2653,E1 2.3467,E2 216.5613} C_DIS
LIN {X -87.8809,Y -111.5016,Z 187,A -121.5528,B 2.4309,C 0.2683,E1 2.3507,E2 214.7582} C_DIS
LIN {X -84.2287,Y -114.2855,Z 187,A -119.6146,B 2.4306,C 0.2708,E1 2.355,E2 212.8081} C_DIS
LIN {X -80.766,Y -116.7587,Z 187,A -117.8085,B 2.4303,C 0.2729,E1 2.3592,E2 210.9895} C_DIS
LIN {X -77.138,Y -119.1863,Z 187,A -116.0542,B 2.4301,C 0.2754,E1 2.3633,E2 209.2362} C_DIS
LIN {X -73.5015,Y -121.4625,Z 187,A -114.211,B 2.4299,C 0.2772,E1 2.3677,E2 207.3772} C_DIS
LIN {X -69.4403,Y -123.8292,Z 187,A -112.1677,B 2.4297,C 0.2788,E1 2.3727,E2 205.313} C_DIS
LIN {X -64.783,Y -126.3264,Z 187,A -110.2283,B 2.4293,C 0.2822,E1 2.3775,E2 203.4006} C_DIS
LIN {X -61.5423,Y -127.9364,Z 187,A -108.6735,B 2.4292,C 0.2833,E1 2.3814,E2 201.8323} C_DIS
LIN {X -58.5031,Y -129.3552,Z 187,A -107.2872,B 2.429,C 0.2845,E1 2.385,E2 200.4412} C_DIS
LIN {X -55.1936,Y -130.8013,Z 187,A -105.8687,B 2.4288,C 0.286,E1 2.3886,E2 199.0279} C_DIS
LIN {X -52.2608,Y -132.0024,Z 187,A -104.511,B 2.4288,C 0.2867,E1 2.3921,E2 197.659} C_DIS
LIN {X -46.6493,Y -134.0855,Z 187,A -101.408,B 2.429,C 0.285,E1 2.4006,E2 194.4577} C_DIS
LIN {X -41.5623,Y -135.7485,Z 187,A -100.0568,B 2.4283,C 0.2907,E1 2.4039,E2 193.2208} C_DIS
LIN {X -37.7623,Y -136.8552,Z 187,A -98.2284,B 2.4283,C 0.2904,E1 2.4089,E2 191.3593} C_DIS
LIN {X -33.4265,Y -137.9775,Z 187,A -96.4016,B 2.4283,C 0.2912,E1 2.4139,E2 189.5293} C_DIS
LIN {X -29.8376,Y -138.7979,Z 187,A -94.9145,B 2.4282,C 0.2918,E1 2.4179,E2 188.0415} C_DIS
LIN {X -26.2614,Y -139.5192,Z 187,A -93.3452,B 2.4282,C 0.2918,E1 2.4223,E2 186.458} C_DIS
LIN {X -22.0042,Y -140.2535,Z 187,A -91.8371,B 2.4279,C 0.2935,E1 2.4263,E2 184.9825} C_DIS
LIN {X -19.2611,Y -140.6585,Z 187,A -90.4699,B 2.4281,C 0.2923,E1 2.4302,E2 183.5798} C_DIS
LIN {X -15.384,Y -141.133,Z 187,A -88.9186,B 2.4281,C 0.2926,E1 2.4345,E2 182.0314} C_DIS
LIN {X -11.0414,Y -141.5407,Z 187,A -87.1348,B 2.4281,C 0.2926,E1 2.4395,E2 180.2436} C_DIS
LIN {X -7.3501,Y -141.7787,Z 187,A -85.7807,B 2.428,C 0.2933,E1 2.4432,E2 178.9085} C_DIS
LIN {X -4.2244,Y -141.9064,Z 187,A -84.4331,B 2.428,C 0.2927,E1 2.4471,E2 177.5482} C_DIS
LIN {X -0.3261,Y -141.9694,Z 187,A -82.8565,B 2.428,C 0.2924,E1 2.4515,E2 175.9704} C_DIS
LIN {X -0.3261,Y -141.9694,Z 187,A -82.8565,B 2.428,C 0.2924,E1 2.4515,E2 175.9704} C_DIS
Enddeposition()
LIN {X 1.0055,Y -142.8642,Z 187,A -82.6748,B 2.4276,C 0.2957,E1 2.4517,E2 175.8685} C_DIS
Startdeposition()
$VEL.CP = VEL_PRINT
LIN {X -1.7502,Y -142.8594,Z 187,A -83.9722,B 2.4274,C 0.2971,E1 2.448,E2 177.1938} C_DIS
LIN {X -5.1483,Y -142.7765,Z 187,A -85.4521,B 2.4274,C 0.298,E1 2.4438,E2 178.6909} C_DIS
LIN {X -9.3262,Y -142.5649,Z 187,A -87.2182,B 2.4272,C 0.2986,E1 2.4388,E2 180.4703} C_DIS
LIN {X -13.4333,Y -142.2358,Z 187,A -88.8379,B 2.4272,C 0.2983,E1 2.4343,E2 182.0859} C_DIS
LIN {X -17.4844,Y -141.7957,Z 187,A -90.376,B 2.4274,C 0.2976,E1 2.4301,E2 183.6112} C_DIS
LIN {X -20.3914,Y -141.4059,Z 187,A -91.6212,B 2.4274,C 0.2978,E1 2.4266,E2 184.8665} C_DIS
LIN {X -24.4163,Y -140.7687,Z 187,A -93.2255,B 2.4274,C 0.2972,E1 2.4222,E2 186.4673} C_DIS
LIN {X -27.8719,Y -140.1247,Z 187,A -94.6376,B 2.4274,C 0.2967,E1 2.4183,E2 187.8802} C_DIS
LIN {X -30.7412,Y -139.5232,Z 187,A -95.9273,B 2.4274,C 0.2969,E1 2.4147,E2 189.1863} C_DIS
LIN {X -34.7031,Y -138.5903,Z 187,A -97.4674,B 2.4276,C 0.2956,E1 2.4105,E2 190.714} C_DIS
LIN {X -38.0888,Y -137.6981,Z 187,A -98.8863,B 2.4276,C 0.2949,E1 2.4067,E2 192.1354} C_DIS
LIN {X -41.3787,Y -136.7456,Z 187,A -100.4047,B 2.4276,C 0.2949,E1 2.4026,E2 193.6746} C_DIS
LIN {X -45.9221,Y -135.2892,Z 187,A -102.2174,B 2.4279,C 0.293,E1 2.3978,E2 195.4736} C_DIS
LIN {X -49.222,Y -134.1237,Z 187,A -103.7773,B 2.4279,C 0.2927,E1 2.3936,E2 197.0559} C_DIS
LIN {X -53.5775,Y -132.4417,Z 187,A -105.6167,B 2.4282,C 0.291,E1 2.3889,E2 198.891} C_DIS
LIN {X -57.3757,Y -130.8429,Z 187,A -107.2105,B 2.4284,C 0.2892,E1 2.3848,E2 200.4768} C_DIS
LIN {X -60.2907,Y -129.524,Z 187,A -108.5468,B 2.4284,C 0.2882,E1 2.3814,E2 201.8207} C_DIS
LIN {X -63.4451,Y -128.0081,Z 187,A -110.041,B 2.4286,C 0.2871,E1 2.3776,E2 203.3279} C_DIS
LIN {X -67.592,Y -125.8698,Z 187,A -111.989,B 2.4288,C 0.2853,E1 2.3727,E2 205.2869} C_DIS
LIN {X -71.6918,Y -123.5807,Z 187,A -113.8701,B 2.4291,C 0.283,E1 2.3681,E2 207.1679} C_DIS
LIN {X -75.4552,Y -121.3193,Z 187,A -115.7249,B 2.4293,C 0.2811,E1 2.3637,E2 209.036} C_DIS
LIN {X -79.3738,Y -118.7926,Z 187,A -117.6602,B 2.4296,C 0.2788,E1 2.3591,E2 210.9805} C_DIS
LIN {X -82.9749,Y -116.3059,Z 187,A -119.4261,B 2.4299,C 0.2763,E1 2.3551,E2 212.7481} C_DIS
LIN {X -86.4998,Y -113.7092,Z 187,A -121.2504,B 2.4301,C 0.2739,E1 2.351,E2 214.5819} C_DIS
LIN {X -89.9551,Y -110.9958,Z 187,A -123.1253,B 2.4304,C 0.2715,E1 2.3468,E2 216.4725} C_DIS
LIN {X -93.3243,Y -108.1779,Z 187,A -124.935,B 2.4307,C 0.2687,E1 2.343,E2 218.2888} C_DIS
LIN {X -96.5904,Y -105.272,Z 187,A -126.7531,B 2.431,C 0.2659,E1 2.3392,E2 220.1158} C_DIS
LIN {X -99.9718,Y -102.0663,Z 187,A -128.6954,B 2.4314,C 0.2628,E1 2.3353,E2 222.0681} C_DIS
LIN {X -103.2752,Y -98.7223,Z 187,A -130.6477,B 2.4317,C 0.2594,E1 2.3314,E2 224.0295} C_DIS
LIN {X -106.2526,Y -95.5108,Z 187,A -132.4486,B 2.4321,C 0.2561,E1 2.328,E2 225.8362} C_DIS
LIN {X -108.9404,Y -92.4331,Z 187,A -134.2039,B 2.4324,C 0.2532,E1 2.3248,E2 227.6074} C_DIS
LIN {X -111.9606,Y -88.7512,Z 187,A -136.1891,B 2.4328,C 0.2495,E1 2.3213,E2 229.6026} C_DIS
LIN {X -114.7434,Y -85.1228,Z 187,A -138.12,B 2.4331,C 0.2459,E1 2.318,E2 231.5464} C_DIS
LIN {X -117.4743,Y -81.3129,Z 187,A -140.1073,B 2.4335,C 0.2421,E1 2.3148,E2 233.5481} C_DIS
LIN {X -120.0818,Y -77.4109,Z 187,A -142.0863,B 2.4339,C 0.2381,E1 2.3117,E2 235.5399} C_DIS
LIN {X -122.5438,Y -73.4508,Z 187,A -143.9922,B 2.4343,C 0.2338,E1 2.309,E2 237.45} C_DIS
LIN {X -124.7361,Y -69.663,Z 187,A -145.8979,B 2.4347,C 0.2301,E1 2.3063,E2 239.3759} C_DIS
LIN {X -126.8159,Y -65.7989,Z 187,A -147.6372,B 2.4351,C 0.2258,E1 2.304,E2 241.1117} C_DIS
LIN {X -128.3934,Y -62.6641,Z 187,A -149.1188,B 2.4354,C 0.2226,E1 2.3022,E2 242.6029} C_DIS
LIN {X -129.7775,Y -59.7425,Z 187,A -150.5173,B 2.4356,C 0.2196,E1 2.3005,E2 244.0148} C_DIS
LIN {X -131.5392,Y -55.7613,Z 187,A -152.4816,B 2.436,C 0.2158,E1 2.2983,E2 246.0082} C_DIS
LIN {X -133.2932,Y -51.4235,Z 187,A -154.3078,B 2.4364,C 0.2109,E1 2.2964,E2 247.8267} C_DIS
LIN {X -134.5124,Y -48.1439,Z 187,A -155.7929,B 2.4367,C 0.2074,E1 2.295,E2 249.3222} C_DIS
LIN {X -135.6569,Y -44.818,Z 187,A -157.2838,B 2.437,C 0.2039,E1 2.2937,E2 250.8234} C_DIS
LIN {X -136.8838,Y -40.9248,Z 187,A -159.1811,B 2.4373,C 0.2003,E1 2.2921,E2 252.7552} C_DIS
LIN {X -138.003,Y -36.9671,Z 187,A -160.7647,B 2.4377,C 0.1957,E1 2.2909,E2 254.3291} C_DIS
LIN {X -138.8337,Y -33.7138,Z 187,A -162.2258,B 2.4379,C 0.1924,E1 2.2899,E2 255.8049} C_DIS
LIN {X -139.624,Y -30.2741,Z 187,A -163.7212,B 2.4382,C 0.1887,E1 2.289,E2 257.3104} C_DIS
LIN {X -140.3524,Y -26.6946,Z 187,A -165.243,B 2.4385,C 0.1848,E1 2.2882,E2 258.8391} C_DIS
LIN {X -141.0581,Y -22.6869,Z 187,A -166.9881,B 2.4388,C 0.1806,E1 2.2873,E2 260.5985} C_DIS
LIN {X -141.5703,Y -19.2277,Z 187,A -168.3881,B 2.4391,C 0.1767,E1 2.2868,E2 261.9974} C_DIS
LIN {X -141.9344,Y -16.3221,Z 187,A -169.8372,B 2.4393,C 0.1742,E1 2.2863,E2 263.4826} C_DIS
LIN {X -142.3901,Y -11.6876,Z 187,A -171.7953,B 2.4397,C 0.1692,E1 2.2858,E2 265.4515} C_DIS
LIN {X -142.6676,Y -7.588,Z 187,A -173.5625,B 2.44,C 0.1649,E1 2.2855,E2 267.2336} C_DIS
LIN {X -142.8396,Y -2.9353,Z 187,A -175.5353,B 2.4403,C 0.1599,E1 2.2853,E2 269.2194} C_DIS
LIN {X -142.8665,Y 0.7733,Z 187,A -177.0578,B 2.4406,C 0.1558,E1 2.2853,E2 270.7456} C_DIS
LIN {X -142.7728,Y 5.2417,Z 187,A -178.9229,B 2.4409,C 0.1509,E1 2.2855,E2 272.6191} C_DIS
LIN {X -142.5645,Y 9.3336,Z 187,A 179.2378,B 2.4411,C 0.1468,E1 2.2858,E2 274.4834} C_DIS
LIN {X -142.2362,Y 13.4291,Z 187,A 177.4947,B 2.4414,C 0.1424,E1 2.2862,E2 276.2378} C_DIS
LIN {X -141.7969,Y 17.4746,Z 187,A 175.8691,B 2.4416,C 0.1379,E1 2.2867,E2 277.8615} C_DIS
LIN {X -141.4072,Y 20.382,Z 187,A 174.5518,B 2.4418,C 0.135,E1 2.2873,E2 279.1966} C_DIS
LIN {X -140.7667,Y 24.4273,Z 187,A 172.8572,B 2.442,C 0.1305,E1 2.288,E2 280.897} C_DIS
LIN {X -140.129,Y 27.8509,Z 187,A 171.3777,B 2.4422,C 0.1269,E1 2.2888,E2 282.3863} C_DIS
LIN {X -139.5278,Y 30.7197,Z 187,A 170.0123,B 2.4424,C 0.1241,E1 2.2896,E2 283.7757} C_DIS
LIN {X -138.5871,Y 34.7154,Z 187,A 168.3864,B 2.4426,C 0.1196,E1 2.2907,E2 285.3978} C_DIS
LIN {X -137.694,Y 38.1035,Z 187,A 166.8983,B 2.4428,C 0.116,E1 2.2918,E2 286.8957} C_DIS
LIN {X -136.7161,Y 41.4749,Z 187,A 165.2936,B 2.4429,C 0.1127,E1 2.2931,E2 288.525} C_DIS
LIN {X -135.2838,Y 45.9385,Z 187,A 163.4172,B 2.4431,C 0.1077,E1 2.2947,E2 290.3997} C_DIS
LIN {X -134.1162,Y 49.243,Z 187,A 161.8363,B 2.4433,C 0.1045,E1 2.2962,E2 292.0023} C_DIS
LIN {X -132.4415,Y 53.5779,Z 187,A 159.8885,B 2.4435,C 0.0999,E1 2.2983,E2 293.9595} C_DIS
LIN {X -130.8458,Y 57.369,Z 187,A 158.2434,B 2.4437,C 0.0956,E1 2.3001,E2 295.6028} C_DIS
LIN {X -129.5296,Y 60.2785,Z 187,A 156.8619,B 2.4437,C 0.0927,E1 2.3017,E2 296.9964} C_DIS
LIN {X -128.0049,Y 63.4516,Z 187,A 155.3504,B 2.4439,C 0.0894,E1 2.3036,E2 298.5197} C_DIS
LIN {X -125.9951,Y 67.3588,Z 187,A 153.4567,B 2.444,C 0.0854,E1 2.306,E2 300.4291} C_DIS
LIN {X -123.8731,Y 71.1865,Z 187,A 151.6025,B 2.4442,C 0.0815,E1 2.3086,E2 302.2947} C_DIS
LIN {X -121.6342,Y 74.9472,Z 187,A 149.7783,B 2.4442,C 0.0775,E1 2.3112,E2 304.1264} C_DIS
LIN {X -119.4382,Y 78.3992,Z 187,A 148.0418,B 2.4444,C 0.074,E1 2.3139,E2 305.874} C_DIS
LIN {X -116.9775,Y 82.0262,Z 187,A 146.1809,B 2.4445,C 0.0703,E1 2.3168,E2 307.7467} C_DIS
LIN {X -114.3492,Y 85.6522,Z 187,A 144.3329,B 2.4446,C 0.0665,E1 2.3199,E2 309.6} C_DIS
LIN {X -111.9138,Y 88.81,Z 187,A 142.5872,B 2.4446,C 0.0635,E1 2.323,E2 311.3631} C_DIS
LIN {X -108.9396,Y 92.4341,Z 187,A 140.733,B 2.4448,C 0.0595,E1 2.3263,E2 313.2127} C_DIS
LIN {X -106.5124,Y 95.2207,Z 187,A 139.0685,B 2.4448,C 0.057,E1 2.3294,E2 314.8992} C_DIS
LIN {X -103.2714,Y 98.7263,Z 187,A 137.0873,B 2.4449,C 0.0535,E1 2.3332,E2 316.8873} C_DIS
LIN {X -99.9813,Y 102.0569,Z 187,A 135.1325,B 2.445,C 0.0502,E1 2.3371,E2 318.8506} C_DIS
LIN {X -96.5976,Y 105.2653,Z 187,A 133.2379,B 2.445,C 0.0468,E1 2.3409,E2 320.7469} C_DIS
LIN {X -93.4162,Y 108.0988,Z 187,A 131.4828,B 2.4451,C 0.044,E1 2.3446,E2 322.5067} C_DIS
LIN {X -90.4125,Y 110.623,Z 187,A 129.7839,B 2.4451,C 0.0417,E1 2.3483,E2 324.2203} C_DIS
LIN {X -86.9811,Y 113.3411,Z 187,A 127.9531,B 2.4452,C 0.0391,E1 2.3524,E2 326.0593} C_DIS
LIN {X -83.2209,Y 116.13,Z 187,A 126.0205,B 2.4452,C 0.0364,E1 2.3568,E2 327.9975} C_DIS
LIN {X -79.3688,Y 118.7959,Z 187,A 124.0895,B 2.4452,C 0.0339,E1 2.3612,E2 329.9338} C_DIS
LIN {X -75.4539,Y 121.3202,Z 187,A 122.1602,B 2.4453,C 0.0315,E1 2.3658,E2 331.8695} C_DIS
LIN {X -71.7045,Y 123.5733,Z 187,A 120.3538,B 2.4453,C 0.0294,E1 2.3702,E2 333.6813} C_DIS
LIN {X -67.6033,Y 125.8637,Z 187,A 118.4588,B 2.4453,C 0.0272,E1 2.3748,E2 335.5764} C_DIS
LIN {X -64.7687,Y 127.3432,Z 187,A 117.1562,B 2.4453,C 0.0258,E1 2.3781,E2 336.8807} C_DIS
LIN {X -61.6072,Y 128.9025,Z 187,A 115.7101,B 2.4454,C 0.0244,E1 2.3817,E2 338.3299} C_DIS
LIN {X -57.8978,Y 130.6116,Z 187,A 114.0109,B 2.4454,C 0.023,E1 2.3861,E2 340.0358} C_DIS
LIN {X -53.591,Y 132.4362,Z 187,A 112.1742,B 2.4454,C 0.021,E1 2.3908,E2 341.8664} C_DIS
LIN {X -49.8025,Y 133.9072,Z 187,A 110.5128,B 2.4454,C 0.0198,E1 2.3951,E2 343.5308} C_DIS
LIN {X -46.5075,Y 135.0869,Z 187,A 109.0827,B 2.4454,C 0.0188,E1 2.3989,E2 344.9634} C_DIS
LIN {X -43.1501,Y 136.1966,Z 187,A 107.5856,B 2.4454,C 0.0181,E1 2.4029,E2 346.4695} C_DIS
LIN {X -39.0882,Y 137.4186,Z 187,A 105.8087,B 2.4454,C 0.0174,E1 2.4077,E2 348.2549} C_DIS
LIN {X -35.2643,Y 138.4478,Z 187,A 104.3161,B 2.4454,C 0.0161,E1 2.4117,E2 349.7348} C_DIS
LIN {X -31.3122,Y 139.3958,Z 187,A 102.6751,B 2.4454,C 0.0153,E1 2.4162,E2 351.3763} C_DIS
LIN {X -28.4486,Y 140.0073,Z 187,A 101.4861,B 2.4454,C 0.0149,E1 2.4195,E2 352.5664} C_DIS
LIN {X -25.0113,Y 140.6622,Z 187,A 100.0167,B 2.4454,C 0.0148,E1 2.4235,E2 354.0434} C_DIS
LIN {X -20.9931,Y 141.3199,Z 187,A 98.4057,B 2.4454,C 0.0142,E1 2.428,E2 355.6509} C_DIS
LIN {X -18.0578,Y 141.7236,Z 187,A 97.247,B 2.4454,C 0.0138,E1 2.4312,E2 356.8053} C_DIS
LIN {X -14.0121,Y 142.1802,Z 187,A 95.494,B 2.4454,C 0.0142,E1 2.4361,E2 358.5724} C_DIS
LIN {X -9.3405,Y 142.564,Z 187,A 93.7031,B 2.4454,C 0.0137,E1 2.4411,E2 360.3515} C_DIS
LIN {X -5.8298,Y 142.7499,Z 187,A 92.2169,B 2.4454,C 0.0141,E1 2.4452,E2 361.8465} C_DIS
LIN {X -1.7565,Y 142.8592,Z 187,A 90.7278,B 2.4454,C 0.0135,E1 2.4494,E2 363.3168} C_DIS
LIN {X 1.1797,Y 142.8644,Z 187,A 89.5187,B 2.4454,C 0.0139,E1 2.4528,E2 364.5294} C_DIS
LIN {X 5.2472,Y 142.7726,Z 187,A 87.8719,B 2.4454,C 0.0144,E1 2.4574,E2 366.1774} C_DIS
LIN {X 9.3322,Y 142.5646,Z 187,A 86.1281,B 2.4454,C 0.0155,E1 2.4623,E2 367.9335} C_DIS
LIN {X 13.9984,Y 142.1815,Z 187,A 84.397,B 2.4454,C 0.0155,E1 2.467,E2 369.6457} C_DIS
LIN {X 17.4806,Y 141.7962,Z 187,A 83.009,B 2.4454,C 0.016,E1 2.4709,E2 371.0311} C_DIS
LIN {X 20.3884,Y 141.4063,Z 187,A 81.7791,B 2.4454,C 0.017,E1 2.4743,E2 372.2672} C_DIS
LIN {X 24.4252,Y 140.7671,Z 187,A 80.2063,B 2.4454,C 0.0176,E1 2.4786,E2 373.8312} C_DIS
LIN {X 27.8667,Y 140.1258,Z 187,A 78.8251,B 2.4454,C 0.0184,E1 2.4824,E2 375.2092} C_DIS
LIN {X 30.7377,Y 139.5239,Z 187,A 77.5652,B 2.4454,C 0.0198,E1 2.4859,E2 376.4793} C_DIS
LIN {X 34.6972,Y 138.5918,Z 187,A 76.0661,B 2.4454,C 0.0203,E1 2.4899,E2 377.9613} C_DIS
LIN {X 38.1024,Y 137.6943,Z 187,A 74.6835,B 2.4454,C 0.0214,E1 2.4936,E2 379.3398} C_DIS
LIN {X 41.4435,Y 136.7257,Z 187,A 73.2061,B 2.4454,C 0.0232,E1 2.4976,E2 380.8273} C_DIS
LIN {X 45.914,Y 135.2919,Z 187,A 71.4694,B 2.4454,C 0.0242,E1 2.5022,E2 382.5453} C_DIS
LIN {X 49.2406,Y 134.117,Z 187,A 69.9461,B 2.4454,C 0.0265,E1 2.5062,E2 384.082} C_DIS
LIN {X 53.585,Y 132.4386,Z 187,A 68.1983,B 2.4454,C 0.0279,E1 2.5108,E2 385.8143} C_DIS
LIN {X 57.3731,Y 130.8441,Z 187,A 66.6791,B 2.4454,C 0.029,E1 2.5146,E2 387.3171} C_DIS
LIN {X 60.2857,Y 129.5263,Z 187,A 65.3538,B 2.4454,C 0.031,E1 2.518,E2 388.6476} C_DIS
LIN {X 63.699,Y 127.8829,Z 187,A 63.9064,B 2.4454,C 0.0326,E1 2.5216,E2 390.0858} C_DIS
LIN {X 67.3375,Y 126.0065,Z 187,A 62.2947,B 2.4453,C 0.0347,E1 2.5256,E2 391.6937} C_DIS
LIN {X 71.1879,Y 123.8723,Z 187,A 60.5623,B 2.4453,C 0.0371,E1 2.5298,E2 393.4218} C_DIS
LIN {X 74.95,Y 121.6324,Z 187,A 58.8819,B 2.4453,C 0.0394,E1 2.5338,E2 395.0925} C_DIS
LIN {X 78.4027,Y 119.4359,Z 187,A 57.2837,B 2.4452,C 0.0417,E1 2.5375,E2 396.6852} C_DIS
LIN {X 82.0264,Y 116.9774,Z 187,A 55.5805,B 2.4452,C 0.0443,E1 2.5415,E2 398.3817} C_DIS
LIN {X 85.2511,Y 114.6478,Z 187,A 53.9913,B 2.4451,C 0.0471,E1 2.545,E2 399.9701} C_DIS
LIN {X 88.81,Y 111.9138,Z 187,A 52.2664,B 2.4451,C 0.0498,E1 2.5488,E2 401.6856} C_DIS
LIN {X 92.4364,Y 108.9376,Z 187,A 50.558,B 2.445,C 0.0521,E1 2.5524,E2 403.3721} C_DIS
LIN {X 95.2909,Y 106.4496,Z 187,A 49.0096,B 2.4449,C 0.0553,E1 2.5557,E2 404.9244} C_DIS
LIN {X 98.7232,Y 103.2744,Z 187,A 47.2063,B 2.4449,C 0.0585,E1 2.5593,E2 406.7187} C_DIS
LIN {X 102.0554,Y 99.9829,Z 187,A 45.4052,B 2.4447,C 0.0618,E1 2.5629,E2 408.5103} C_DIS
LIN {X 105.2656,Y 96.5973,Z 187,A 43.6574,B 2.4447,C 0.0648,E1 2.5662,E2 410.2425} C_DIS
LIN {X 108.1822,Y 93.3193,Z 187,A 42.0193,B 2.4446,C 0.0676,E1 2.5692,E2 411.8653} C_DIS
LIN {X 110.618,Y 90.4187,Z 187,A 40.4924,B 2.4445,C 0.0711,E1 2.5719,E2 413.3936} C_DIS
LIN {X 113.3367,Y 86.9869,Z 187,A 38.7861,B 2.4444,C 0.0747,E1 2.5748,E2 415.0938} C_DIS
LIN {X 116.1255,Y 83.2271,Z 187,A 37.002,B 2.4443,C 0.0783,E1 2.5777,E2 416.8664} C_DIS
LIN {X 118.7945,Y 79.371,Z 187,A 35.2173,B 2.4441,C 0.082,E1 2.5805,E2 418.6392} C_DIS
LIN {X 121.171,Y 75.6935,Z 187,A 33.5313,B 2.4441,C 0.0856,E1 2.583,E2 420.3167} C_DIS
LIN {X 123.4343,Y 71.9446,Z 187,A 31.8469,B 2.4439,C 0.0894,E1 2.5854,E2 421.9924} C_DIS
LIN {X 125.5809,Y 68.1279,Z 187,A 30.18,B 2.4438,C 0.093,E1 2.5877,E2 423.6482} C_DIS
LIN {X 127.352,Y 64.7516,Z 187,A 28.7918,B 2.4437,C 0.0957,E1 2.5894,E2 425.0185} C_DIS
LIN {X 128.901,Y 61.6103,Z 187,A 27.4537,B 2.4435,C 0.0987,E1 2.591,E2 426.3485} C_DIS
LIN {X 130.6132,Y 57.894,Z 187,A 25.8722,B 2.4434,C 0.1024,E1 2.5929,E2 427.9229} C_DIS
LIN {X 132.4396,Y 53.5826,Z 187,A 24.1611,B 2.4432,C 0.1059,E1 2.5947,E2 429.6129} C_DIS
LIN {X 133.9135,Y 49.7858,Z 187,A 22.6096,B 2.4431,C 0.1096,E1 2.5962,E2 431.1544} C_DIS
LIN {X 135.0986,Y 46.4738,Z 187,A 21.2741,B 2.4429,C 0.1127,E1 2.5974,E2 432.4806} C_DIS
LIN {X 136.1977,Y 43.1468,Z 187,A 19.8834,B 2.4428,C 0.1163,E1 2.5986,E2 433.87} C_DIS
LIN {X 137.5419,Y 38.6471,Z 187,A 18.1586,B 2.4426,C 0.1201,E1 2.6,E2 435.5749} C_DIS
LIN {X 138.4468,Y 35.2682,Z 187,A 16.8304,B 2.4424,C 0.1232,E1 2.6009,E2 436.8939} C_DIS
LIN {X 139.3953,Y 31.3142,Z 187,A 15.2921,B 2.4422,C 0.1269,E1 2.6019,E2 438.4209} C_DIS
LIN {X 140.0074,Y 28.4485,Z 187,A 14.1758,B 2.4421,C 0.1296,E1 2.6025,E2 439.5299} C_DIS
LIN {X 140.7627,Y 24.4494,Z 187,A 12.6397,B 2.4419,C 0.1333,E1 2.6033,E2 441.0542} C_DIS
LIN {X 141.3242,Y 20.9632,Z 187,A 11.2793,B 2.4417,C 0.1368,E1 2.6038,E2 442.408} C_DIS
LIN {X 141.7235,Y 18.0589,Z 187,A 10.1899,B 2.4416,C 0.1393,E1 2.6042,E2 443.4866} C_DIS
LIN {X 142.1801,Y 14.0129,Z 187,A 8.5374,B 2.4413,C 0.144,E1 2.6047,E2 445.1426} C_DIS
LIN {X 142.5647,Y 9.3298,Z 187,A 6.8409,B 2.4411,C 0.1477,E1 2.6051,E2 446.8152} C_DIS
LIN {X 142.7722,Y 5.2587,Z 187,A 5.2288,B 2.4408,C 0.1521,E1 2.6053,E2 448.4252} C_DIS
LIN {X 142.8651,Y 1.0367,Z 187,A 3.6531,B 2.4406,C 0.1558,E1 2.6053,E2 449.9861} C_DIS
LIN {X 142.8396,Y -2.9379,Z 187,A 2.0876,B 2.4403,C 0.16,E1 2.6053,E2 451.5489} C_DIS
LIN {X 142.6965,Y -7.0133,Z 187,A 0.5782,B 2.4401,C 0.1635,E1 2.6051,E2 453.0424} C_DIS
LIN {X 142.3903,Y -11.686,Z 187,A -1.1289,B 2.4398,C 0.1672,E1 2.6048,E2 454.7278} C_DIS
LIN {X 141.9995,Y -15.741,Z 187,A -2.6575,B 2.4395,C 0.1709,E1 2.6043,E2 456.2433} C_DIS
LIN {X 141.5727,Y -19.2098,Z 187,A -3.9553,B 2.4393,C 0.1739,E1 2.6039,E2 457.5281} C_DIS
LIN {X 141.0562,Y -22.6981,Z 187,A -5.3404,B 2.4391,C 0.1776,E1 2.6033,E2 458.9102} C_DIS
LIN {X 140.4569,Y -26.1482,Z 187,A -6.6658,B 2.4388,C 0.1808,E1 2.6026,E2 460.2259} C_DIS
LIN {X 139.7735,Y -29.5818,Z 187,A -7.8896,B 2.4387,C 0.183,E1 2.602,E2 461.4262} C_DIS
LIN {X 139.0039,Y -33.0079,Z 187,A -9.323,B 2.4384,C 0.1871,E1 2.6011,E2 462.8641} C_DIS
LIN {X 138.1539,Y -36.401,Z 187,A -10.6549,B 2.4381,C 0.1903,E1 2.6001,E2 464.1873} C_DIS
LIN {X 137.2172,Y -39.7861,Z 187,A -11.9814,B 2.4379,C 0.1935,E1 2.5991,E2 465.5036} C_DIS
LIN {X 136.0298,Y -43.6724,Z 187,A -13.5838,B 2.4375,C 0.1976,E1 2.5978,E2 467.1036} C_DIS
LIN {X 134.7169,Y -47.5747,Z 187,A -15.0924,B 2.4373,C 0.2008,E1 2.5965,E2 468.594} C_DIS
LIN {X 133.3649,Y -51.2389,Z 187,A -16.7224,B 2.4369,C 0.2055,E1 2.5948,E2 470.2339} C_DIS
LIN {X 131.5391,Y -55.7615,Z 187,A -18.4367,B 2.4366,C 0.2085,E1 2.593,E2 471.9166} C_DIS
LIN {X 130.3736,Y -58.4297,Z 187,A -19.5811,B 2.4364,C 0.2114,E1 2.5918,E2 473.0586} C_DIS
LIN {X 128.7724,Y -61.8795,Z 187,A -20.9914,B 2.4361,C 0.2143,E1 2.5901,E2 474.4543} C_DIS
LIN {X 126.9521,Y -65.5371,Z 187,A -22.5898,B 2.4358,C 0.2181,E1 2.5881,E2 476.0486} C_DIS
LIN {X 125.0338,Y -69.1262,Z 187,A -24.1861,B 2.4354,C 0.2219,E1 2.586,E2 477.6412} C_DIS
LIN {X 122.8457,Y -72.9443,Z 187,A -25.8737,B 2.4351,C 0.2256,E1 2.5836,E2 479.3196} C_DIS
LIN {X 120.5523,Y -76.6759,Z 187,A -27.5116,B 2.4348,C 0.2289,E1 2.5812,E2 480.9425} C_DIS
LIN {X 118.3016,Y -80.1037,Z 187,A -29.1042,B 2.4345,C 0.2324,E1 2.5787,E2 482.5292} C_DIS
LIN {X 115.6255,Y -83.9203,Z 187,A -30.8912,B 2.4341,C 0.2361,E1 2.5758,E2 484.3063} C_DIS
LIN {X 112.9937,Y -87.4317,Z 187,A -32.5697,B 2.4338,C 0.2395,E1 2.573,E2 485.9749} C_DIS
LIN {X 110.0453,Y -91.1148,Z 187,A -34.3329,B 2.4335,C 0.2427,E1 2.5699,E2 487.7217} C_DIS
LIN {X 107.207,Y -94.4383,Z 187,A -36.0166,B 2.4331,C 0.2459,E1 2.5669,E2 489.3972} C_DIS
LIN {X 104.2708,Y -97.671,Z 187,A -37.7487,B 2.4328,C 0.2496,E1 2.5636,E2 491.128} C_DIS
LIN {X 101.036,Y -101.0138,Z 187,A -39.542,B 2.4324,C 0.2529,E1 2.5601,E2 492.9128} C_DIS
LIN {X 97.9008,Y -104.0545,Z 187,A -41.1501,B 2.4322,C 0.2553,E1 2.5569,E2 494.5022} C_DIS
LIN {X 94.6692,Y -107.0028,Z 187,A -42.802,B 2.4319,C 0.2579,E1 2.5535,E2 496.1412} C_DIS
LIN {X 91.988,Y -109.3166,Z 187,A -44.2128,B 2.4316,C 0.2606,E1 2.5505,E2 497.5518} C_DIS
LIN {X 88.6002,Y -112.0807,Z 187,A -45.909,B 2.4313,C 0.2634,E1 2.5468,E2 499.2414} C_DIS
LIN {X 85.1286,Y -114.739,Z 187,A -47.6423,B 2.431,C 0.2665,E1 2.5429,E2 500.9732} C_DIS
LIN {X 81.3135,Y -117.4739,Z 187,A -49.4628,B 2.4307,C 0.2693,E1 2.5388,E2 502.7864} C_DIS
LIN {X 77.4358,Y -120.0656,Z 187,A -51.2201,B 2.4304,C 0.2715,E1 2.5347,E2 504.5293} C_DIS
LIN {X 73.7305,Y -122.3754,Z 187,A -52.8957,B 2.4302,C 0.2738,E1 2.5307,E2 506.1956} C_DIS
LIN {X 69.9117,Y -124.5963,Z 187,A -54.6184,B 2.4299,C 0.2761,E1 2.5266,E2 507.9127} C_DIS
LIN {X 66.3218,Y -126.5414,Z 187,A -56.1689,B 2.4297,C 0.2779,E1 2.5228,E2 509.452} C_DIS
LIN {X 62.9213,Y -128.2665,Z 187,A -57.6303,B 2.4295,C 0.2795,E1 2.5191,E2 510.9051} C_DIS
LIN {X 59.7685,Y -129.7654,Z 187,A -59.0482,B 2.4293,C 0.2815,E1 2.5155,E2 512.3264} C_DIS
LIN {X 55.7635,Y -131.5383,Z 187,A -60.8688,B 2.429,C 0.2843,E1 2.5108,E2 514.1574} C_DIS
LIN {X 51.956,Y -133.0862,Z 187,A -62.4249,B 2.4288,C 0.2856,E1 2.5068,E2 515.7016} C_DIS
LIN {X 48.1434,Y -134.5126,Z 187,A -63.9287,B 2.4287,C 0.2865,E1 2.5029,E2 517.1883} C_DIS
LIN {X 44.8319,Y -135.6523,Z 187,A -65.3042,B 2.4285,C 0.2878,E1 2.4993,E2 518.5607} C_DIS
LIN {X 40.9178,Y -136.8858,Z 187,A -67.0652,B 2.4282,C 0.2903,E1 2.4945,E2 520.339} C_DIS
LIN {X 36.9568,Y -138.0057,Z 187,A -68.5349,B 2.4282,C 0.2905,E1 2.4906,E2 521.7841} C_DIS
LIN {X 33.5637,Y -138.8699,Z 187,A -69.9754,B 2.428,C 0.292,E1 2.4867,E2 523.2307} C_DIS
LIN {X 29.5926,Y -139.7712,Z 187,A -71.4688,B 2.428,C 0.2923,E1 2.4827,E2 524.7054} C_DIS
LIN {X 26.7194,Y -140.3477,Z 187,A -72.6768,B 2.4279,C 0.2934,E1 2.4793,E2 525.9186} C_DIS
LIN {X 22.708,Y -141.0546,Z 187,A -74.2958,B 2.4277,C 0.2944,E1 2.4749,E2 527.5366} C_DIS
LIN {X 19.2451,Y -141.568,Z 187,A -75.6118,B 2.4277,C 0.2946,E1 2.4713,E2 528.841} C_DIS
LIN {X 16.3161,Y -141.9351,Z 187,A -76.9656,B 2.4275,C 0.2964,E1 2.4674,E2 530.2194} C_DIS
LIN {X 11.6911,Y -142.3898,Z 187,A -78.7859,B 2.4275,C 0.2969,E1 2.4624,E2 532.0346} C_DIS
LIN {X 7.5882,Y -142.6676,Z 187,A -80.3407,B 2.4275,C 0.2969,E1 2.4581,E2 533.5769} C_DIS
LIN {X 3.5047,Y -142.8264,Z 187,A -81.9429,B 2.4275,C 0.2972,E1 2.4536,E2 535.1747} C_DIS
LIN {X 1.0055,Y -142.8642,Z 187,A -82.6746,B 2.4275,C 0.2957,E1 2.4517,E2 535.8685} C_DIS
Enddeposition()
LIN {X 0.9694,Y -133.9063,Z 188,A -82.849,B 2.3884,C 0.2824,E1 2.4113,E2 535.7766} C_DIS
Startdeposition()
$VEL.CP = VEL_PRINT
LIN {X 3.2695,Y -133.8722,Z 188,A -81.5417,B 2.3886,C 0.2802,E1 2.4151,E2 534.4263} C_DIS
LIN {X 7.3472,Y -133.711,Z 188,A -79.6293,B 2.3888,C 0.2787,E1 2.4205,E2 532.491} C_DIS
LIN {X 11.6054,Y -133.4078,Z 188,A -78.0194,B 2.3888,C 0.2792,E1 2.4249,E2 530.9087} C_DIS
LIN {X 14.8682,Y -133.0843,Z 188,A -76.5785,B 2.3888,C 0.2783,E1 2.4289,E2 529.4621} C_DIS
LIN {X 18.0186,Y -132.6948,Z 188,A -75.2723,B 2.3889,C 0.2778,E1 2.4326,E2 528.162} C_DIS
LIN {X 21.5368,Y -132.1689,Z 188,A -73.8139,B 2.3889,C 0.2773,E1 2.4366,E2 526.7111} C_DIS
LIN {X 24.7064,Y -131.6129,Z 188,A -72.4371,B 2.3891,C 0.2763,E1 2.4404,E2 525.3335} C_DIS
LIN {X 27.8487,Y -130.9839,Z 188,A -71.0665,B 2.3892,C 0.2753,E1 2.4441,E2 523.9621} C_DIS
LIN {X 31.0515,Y -130.2616,Z 188,A -69.6871,B 2.3893,C 0.2743,E1 2.4479,E2 522.5852} C_DIS
LIN {X 34.2484,Y -129.4576,Z 188,A -68.3037,B 2.3895,C 0.2732,E1 2.4516,E2 521.2045} C_DIS
LIN {X 37.4149,Y -128.5781,Z 188,A -66.9267,B 2.3895,C 0.272,E1 2.4553,E2 519.8304} C_DIS
LIN {X 40.5573,Y -127.6216,Z 188,A -65.5512,B 2.3897,C 0.2708,E1 2.459,E2 518.458} C_DIS
LIN {X 43.6885,Y -126.5839,Z 188,A -64.1722,B 2.3899,C 0.2695,E1 2.4626,E2 517.0823} C_DIS
LIN {X 47.552,Y -125.1851,Z 188,A -62.3095,B 2.3902,C 0.2668,E1 2.4675,E2 515.2047} C_DIS
LIN {X 51.2366,Y -123.7218,Z 188,A -60.8049,B 2.3902,C 0.266,E1 2.4714,E2 513.7242} C_DIS
LIN {X 54.247,Y -122.4319,Z 188,A -59.4348,B 2.3904,C 0.2644,E1 2.4749,E2 512.3572} C_DIS
LIN {X 57.2519,Y -121.0561,Z 188,A -58.0657,B 2.3906,C 0.2628,E1 2.4783,E2 510.9931} C_DIS
LIN {X 60.3191,Y -119.5572,Z 188,A -56.6493,B 2.3908,C 0.2611,E1 2.4819,E2 509.5814} C_DIS
LIN {X 63.1244,Y -118.1018,Z 188,A -55.3363,B 2.391,C 0.2594,E1 2.4851,E2 508.2727} C_DIS
LIN {X 66.0174,Y -116.5096,Z 188,A -53.965,B 2.3912,C 0.2575,E1 2.4885,E2 506.9058} C_DIS
LIN {X 68.8513,Y -114.8575,Z 188,A -52.587,B 2.3914,C 0.2555,E1 2.4918,E2 505.5301} C_DIS
LIN {X 72.2893,Y -112.7249,Z 188,A -50.7943,B 2.3918,C 0.2522,E1 2.496,E2 503.7281} C_DIS
LIN {X 75.8537,Y -110.3579,Z 188,A -49.1639,B 2.3919,C 0.2506,E1 2.4998,E2 502.1225} C_DIS
LIN {X 78.5341,Y -108.4667,Z 188,A -47.8132,B 2.3921,C 0.2485,E1 2.5028,E2 500.7777} C_DIS
LIN {X 81.721,Y -106.087,Z 188,A -46.168,B 2.3924,C 0.2458,E1 2.5065,E2 499.1386} C_DIS
LIN {X 84.3154,Y -104.0367,Z 188,A -44.7998,B 2.3927,C 0.2435,E1 2.5094,E2 497.7754} C_DIS
LIN {X 87.4502,Y -101.4154,Z 188,A -43.122,B 2.3929,C 0.2407,E1 2.513,E2 496.1055} C_DIS
LIN {X 90.4929,Y -98.7102,Z 188,A -41.3285,B 2.3933,C 0.2368,E1 2.5167,E2 494.3039} C_DIS
LIN {X 93.9347,Y -95.4409,Z 188,A -39.4789,B 2.3936,C 0.234,E1 2.5204,E2 492.4764} C_DIS
LIN {X 96.943,Y -92.3835,Z 188,A -37.6229,B 2.394,C 0.23,E1 2.524,E2 490.6163} C_DIS
LIN {X 99.8237,Y -89.2629,Z 188,A -35.8794,B 2.3943,C 0.2266,E1 2.5273,E2 488.8809} C_DIS
LIN {X 102.9608,Y -85.6258,Z 188,A -34.0467,B 2.3946,C 0.2238,E1 2.5305,E2 487.0756} C_DIS
LIN {X 105.0977,Y -82.9893,Z 188,A -32.5325,B 2.3949,C 0.22,E1 2.5332,E2 485.5522} C_DIS
LIN {X 107.5468,Y -79.7896,Z 188,A -31.0226,B 2.3951,C 0.2177,E1 2.5357,E2 484.0687} C_DIS
LIN {X 109.4613,Y -77.1418,Z 188,A -29.5825,B 2.3955,C 0.2141,E1 2.538,E2 482.6221} C_DIS
LIN {X 111.4142,Y -74.2934,Z 188,A -28.3096,B 2.3956,C 0.2122,E1 2.54,E2 481.3745} C_DIS
LIN {X 113.1363,Y -71.6439,Z 188,A -26.9764,B 2.3959,C 0.2091,E1 2.542,E2 480.0427} C_DIS
LIN {X 114.9204,Y -68.7457,Z 188,A -25.6009,B 2.3962,C 0.2061,E1 2.544,E2 478.6765} C_DIS
LIN {X 116.5823,Y -65.8886,Z 188,A -24.2957,B 2.3964,C 0.2035,E1 2.5458,E2 477.3842} C_DIS
LIN {X 118.0029,Y -63.3085,Z 188,A -23.0252,B 2.3967,C 0.2003,E1 2.5475,E2 476.1114} C_DIS
LIN {X 119.8833,Y -59.6683,Z 188,A -21.5347,B 2.3969,C 0.1979,E1 2.5493,E2 474.6533} C_DIS
LIN {X 121.1089,Y -57.1414,Z 188,A -20.266,B 2.3972,C 0.1943,E1 2.5509,E2 473.3751} C_DIS
LIN {X 122.4731,Y -54.1551,Z 188,A -18.8403,B 2.3975,C 0.1905,E1 2.5525,E2 471.9456} C_DIS
LIN {X 123.7681,Y -51.1257,Z 188,A -17.6014,B 2.3976,C 0.1882,E1 2.5538,E2 470.7275} C_DIS
LIN {X 125.1532,Y -47.6371,Z 188,A -16.1213,B 2.3979,C 0.185,E1 2.5553,E2 469.2623} C_DIS
LIN {X 126.0821,Y -45.1169,Z 188,A -14.8561,B 2.3982,C 0.1809,E1 2.5565,E2 467.9814} C_DIS
LIN {X 127.6548,Y -40.4534,Z 188,A -13.0022,B 2.3985,C 0.1774,E1 2.5581,E2 466.1582} C_DIS
LIN {X 128.6078,Y -37.3134,Z 188,A -11.651,B 2.3987,C 0.174,E1 2.5592,E2 464.8126} C_DIS
LIN {X 129.4894,Y -34.1292,Z 188,A -10.3393,B 2.3989,C 0.171,E1 2.5601,E2 463.5129} C_DIS
LIN {X 130.3835,Y -30.5427,Z 188,A -8.8696,B 2.3992,C 0.1676,E1 2.5611,E2 462.0563} C_DIS
LIN {X 131.0093,Y -27.7312,Z 188,A -7.5742,B 2.3994,C 0.1637,E1 2.5618,E2 460.7521} C_DIS
LIN {X 131.6504,Y -24.5104,Z 188,A -6.3584,B 2.3996,C 0.1614,E1 2.5625,E2 459.5593} C_DIS
LIN {X 132.2125,Y -21.2755,Z 188,A -4.9764,B 2.3998,C 0.1576,E1 2.5631,E2 458.1792} C_DIS
LIN {X 132.7301,Y -17.7497,Z 188,A -3.652,B 2.4,C 0.1551,E1 2.5636,E2 456.8791} C_DIS
LIN {X 133.0958,Y -14.7615,Z 188,A -2.3365,B 2.4003,C 0.1512,E1 2.564,E2 455.5592} C_DIS
LIN {X 133.4281,Y -11.365,Z 188,A -1.0091,B 2.4004,C 0.1483,E1 2.5644,E2 454.2476} C_DIS
LIN {X 133.6799,Y -7.8773,Z 188,A 0.394,B 2.4006,C 0.1448,E1 2.5646,E2 452.8553} C_DIS
LIN {X 133.8254,Y -4.8124,Z 188,A 1.6413,B 2.4008,C 0.1417,E1 2.5648,E2 451.6153} C_DIS
LIN {X 133.905,Y -1.4927,Z 188,A 2.941,B 2.401,C 0.1387,E1 2.5648,E2 450.33} C_DIS
LIN {X 133.9004,Y 1.7705,Z 188,A 4.3064,B 2.4012,C 0.1351,E1 2.5648,E2 448.9676} C_DIS
LIN {X 133.8209,Y 4.929,Z 188,A 5.6319,B 2.4014,C 0.1315,E1 2.5647,E2 447.6445} C_DIS
LIN {X 133.652,Y 8.329,Z 188,A 6.9554,B 2.4016,C 0.1285,E1 2.5645,E2 446.3368} C_DIS
LIN {X 133.4082,Y 11.601,Z 188,A 8.2932,B 2.4018,C 0.1251,E1 2.5642,E2 445.0065} C_DIS
LIN {X 133.0824,Y 14.8866,Z 188,A 9.6236,B 2.4019,C 0.1218,E1 2.5638,E2 443.6854} C_DIS
LIN {X 132.6381,Y 18.4284,Z 188,A 10.9935,B 2.4021,C 0.1189,E1 2.5633,E2 442.3343} C_DIS
LIN {X 132.1493,Y 21.6538,Z 188,A 12.3244,B 2.4022,C 0.1155,E1 2.5627,E2 441.0107} C_DIS
LIN {X 131.6271,Y 24.6324,Z 188,A 13.6261,B 2.4024,C 0.1119,E1 2.5621,E2 439.7074} C_DIS
LIN {X 130.8511,Y 28.4642,Z 188,A 15.0744,B 2.4025,C 0.1091,E1 2.5613,E2 438.2859} C_DIS
LIN {X 130.2589,Y 31.0624,Z 188,A 16.2808,B 2.4027,C 0.1055,E1 2.5605,E2 437.0708} C_DIS
LIN {X 129.4576,Y 34.2482,Z 188,A 17.6091,B 2.4028,C 0.1023,E1 2.5596,E2 435.7514} C_DIS
LIN {X 128.4962,Y 37.6945,Z 188,A 18.9995,B 2.403,C 0.0993,E1 2.5585,E2 434.3775} C_DIS
LIN {X 127.6203,Y 40.5615,Z 188,A 20.2697,B 2.403,C 0.0959,E1 2.5575,E2 433.1083} C_DIS
LIN {X 126.4092,Y 44.1921,Z 188,A 21.8453,B 2.4033,C 0.092,E1 2.5561,E2 431.5396} C_DIS
LIN {X 124.9421,Y 48.1843,Z 188,A 23.545,B 2.4033,C 0.0882,E1 2.5544,E2 429.8539} C_DIS
LIN {X 123.7176,Y 51.2466,Z 188,A 24.8775,B 2.4035,C 0.0851,E1 2.553,E2 428.5305} C_DIS
LIN {X 122.424,Y 54.2647,Z 188,A 26.208,B 2.4036,C 0.082,E1 2.5515,E2 427.2086} C_DIS
LIN {X 121.0572,Y 57.2498,Z 188,A 27.5387,B 2.4037,C 0.079,E1 2.55,E2 425.8864} C_DIS
LIN {X 119.5574,Y 60.3187,Z 188,A 28.9261,B 2.4038,C 0.0759,E1 2.5483,E2 424.5075} C_DIS
LIN {X 118.0997,Y 63.1284,Z 188,A 30.2129,B 2.4039,C 0.073,E1 2.5466,E2 423.2286} C_DIS
LIN {X 116.517,Y 66.0045,Z 188,A 31.5867,B 2.4039,C 0.0698,E1 2.5447,E2 421.858} C_DIS
LIN {X 114.8583,Y 68.8499,Z 188,A 32.9181,B 2.4041,C 0.0669,E1 2.5428,E2 420.5357} C_DIS
LIN {X 113.0732,Y 71.7438,Z 188,A 34.2624,B 2.4041,C 0.0642,E1 2.5409,E2 419.2044} C_DIS
LIN {X 111.2831,Y 74.4898,Z 188,A 35.6112,B 2.4042,C 0.0613,E1 2.5388,E2 417.8617} C_DIS
LIN {X 109.4155,Y 77.2068,Z 188,A 37.068,B 2.4043,C 0.0576,E1 2.5364,E2 416.3989} C_DIS
LIN {X 107.4866,Y 79.8704,Z 188,A 38.4115,B 2.4043,C 0.0548,E1 2.5342,E2 415.0628} C_DIS
LIN {X 105.0582,Y 83.0397,Z 188,A 39.9316,B 2.4044,C 0.0524,E1 2.5317,E2 413.565} C_DIS
LIN {X 102.9523,Y 85.6361,Z 188,A 41.434,B 2.4045,C 0.0486,E1 2.529,E2 412.0537} C_DIS
LIN {X 100.2794,Y 88.7507,Z 188,A 42.969,B 2.4045,C 0.0465,E1 2.5262,E2 410.545} C_DIS
LIN {X 97.5544,Y 91.7378,Z 188,A 44.6332,B 2.4046,C 0.0433,E1 2.5231,E2 408.8885} C_DIS
LIN {X 94.6902,Y 94.692,Z 188,A 46.4577,B 2.4046,C 0.0391,E1 2.5195,E2 407.0561} C_DIS
LIN {X 91.7387,Y 97.5535,Z 188,A 48.1354,B 2.4047,C 0.0362,E1 2.5161,E2 405.3879} C_DIS
LIN {X 88.6586,Y 100.3608,Z 188,A 49.8456,B 2.4047,C 0.0332,E1 2.5125,E2 403.6863} C_DIS
LIN {X 85.5414,Y 103.0307,Z 188,A 51.5272,B 2.4048,C 0.0304,E1 2.509,E2 402.0135} C_DIS
LIN {X 82.392,Y 105.5668,Z 188,A 53.0682,B 2.4048,C 0.0285,E1 2.5056,E2 400.495} C_DIS
LIN {X 79.7794,Y 107.5544,Z 188,A 54.4347,B 2.4048,C 0.0263,E1 2.5026,E2 399.1329} C_DIS
LIN {X 76.8924,Y 109.6372,Z 188,A 55.8527,B 2.4048,C 0.0244,E1 2.4994,E2 397.7275} C_DIS
LIN {X 74.2954,Y 111.4129,Z 188,A 57.1971,B 2.4049,C 0.0221,E1 2.4963,E2 396.3833} C_DIS
LIN {X 71.6388,Y 113.1396,Z 188,A 58.5171,B 2.4049,C 0.0201,E1 2.4932,E2 395.0675} C_DIS
LIN {X 68.7435,Y 114.9217,Z 188,A 59.9982,B 2.4049,C 0.0177,E1 2.4896,E2 393.5834} C_DIS
LIN {X 65.9119,Y 116.5692,Z 188,A 61.2525,B 2.4049,C 0.0165,E1 2.4866,E2 392.3466} C_DIS
LIN {X 63.146,Y 118.0902,Z 188,A 62.5938,B 2.4049,C 0.0146,E1 2.4833,E2 391.0065} C_DIS
LIN {X 59.832,Y 119.8026,Z 188,A 64.058,B 2.4049,C 0.0132,E1 2.4797,E2 389.558} C_DIS
LIN {X 57.1475,Y 121.106,Z 188,A 65.3658,B 2.4049,C 0.0113,E1 2.4764,E2 388.2467} C_DIS
LIN {X 54.1511,Y 122.4748,Z 188,A 66.7356,B 2.4049,C 0.0097,E1 2.4729,E2 386.8818} C_DIS
LIN {X 51.133,Y 123.765,Z 188,A 68.1029,B 2.4049,C 0.0083,E1 2.4694,E2 385.5191} C_DIS
LIN {X 48.0839,Y 124.9811,Z 188,A 69.4615,B 2.405,C 0.0069,E1 2.4659,E2 384.1661} C_DIS
LIN {X 44.6762,Y 126.241,Z 188,A 70.9886,B 2.405,C 0.0054,E1 2.4619,E2 382.6425} C_DIS
LIN {X 42.0212,Y 127.1473,Z 188,A 72.1625,B 2.405,C 0.0043,E1 2.4588,E2 381.472} C_DIS
LIN {X 38.7999,Y 128.1673,Z 188,A 73.5719,B 2.405,C 0.0031,E1 2.455,E2 380.0671} C_DIS
LIN {X 35.7126,Y 129.0616,Z 188,A 74.9273,B 2.405,C 0.0019,E1 2.4514,E2 378.7144} C_DIS
LIN {X 32.5372,Y 129.8986,Z 188,A 76.306,B 2.405,C 0.0009,E1 2.4476,E2 377.3392} C_DIS
LIN {X 29.3401,Y 130.6582,Z 188,A 77.6866,B 2.405,C -0.0001,E1 2.4439,E2 375.962} C_DIS
LIN {X 26.1282,Y 131.3386,Z 188,A 79.1937,B 2.405,C -0.0017,E1 2.4397,E2 374.4432} C_DIS
LIN {X 22.8954,Y 131.9412,Z 188,A 80.4518,B 2.405,C -0.0017,E1 2.4363,E2 373.203} C_DIS
LIN {X 19.5252,Y 132.4813,Z 188,A 81.8762,B 2.405,C -0.0024,E1 2.4324,E2 371.7833} C_DIS
LIN {X 16.3932,Y 132.9051,Z 188,A 83.3776,B 2.405,C -0.0039,E1 2.4282,E2 370.265} C_DIS
LIN {X 13.1294,Y 133.2664,Z 188,A 84.668,B 2.405,C -0.0039,E1 2.4246,E2 368.9884} C_DIS
LIN {X 9.8574,Y 133.548,Z 188,A 86.0292,B 2.405,C -0.0043,E1 2.4208,E2 367.6329} C_DIS
LIN {X 6.4599,Y 133.7556,Z 188,A 87.5395,B 2.405,C -0.005,E1 2.4166,E2 366.1168} C_DIS
LIN {X 3.2861,Y 133.8717,Z 188,A 88.8156,B 2.405,C -0.005,E1 2.4131,E2 364.851} C_DIS
LIN {X 0.0054,Y 133.9134,Z 188,A 90.2831,B 2.405,C -0.0055,E1 2.4089,E2 363.3766} C_DIS
LIN {X -3.2778,Y 133.8719,Z 188,A 91.639,B 2.405,C -0.0055,E1 2.4051,E2 362.0269} C_DIS
LIN {X -6.6809,Y 133.7445,Z 188,A 93.0814,B 2.405,C -0.0055,E1 2.4011,E2 360.5869} C_DIS
LIN {X -9.8617,Y 133.5477,Z 188,A 94.4569,B 2.405,C -0.0055,E1 2.3973,E2 359.2106} C_DIS
LIN {X -13.2446,Y 133.2554,Z 188,A 95.8902,B 2.405,C -0.0052,E1 2.3933,E2 357.7803} C_DIS
LIN {X -16.5057,Y 132.8916,Z 188,A 97.2928,B 2.405,C -0.005,E1 2.3894,E2 356.3786} C_DIS
LIN {X -20.1256,Y 132.3907,Z 188,A 98.7686,B 2.405,C -0.0042,E1 2.3853,E2 354.9138} C_DIS
LIN {X -23.0166,Y 131.9195,Z 188,A 100.1523,B 2.405,C -0.0044,E1 2.3815,E2 353.5155} C_DIS
LIN {X -26.2458,Y 131.3147,Z 188,A 101.6367,B 2.405,C -0.0043,E1 2.3774,E2 352.0227} C_DIS
LIN {X -29.4578,Y 130.6313,Z 188,A 102.9826,B 2.405,C -0.0034,E1 2.3737,E2 350.6844} C_DIS
LIN {X -32.651,Y 129.8697,Z 188,A 104.4017,B 2.405,C -0.0027,E1 2.3699,E2 349.2643} C_DIS
Enddeposition()
END
